// ======================================================
// STORE FLAGS
// ======================================================
GVL_CONFIG_VALIDATION.G_Config_Valid := NOT L_Config_Error;
GVL_CONFIG_VALIDATION.G_Config_Critical_Error := L_Config_Error;
GVL_CONFIG_VALIDATION.G_Config_Last_Update_MS := GVL_STATUS.G_System_Time_MS;

IF L_Config_Error THEN
    GVL_CONFIG_VALIDATION.G_Config_Last_Error_Text := 'CONFIG VALIDATION ERROR';
    GVL_STATUS.G_System_Mode_Text := 'CONFIG ERROR';
ELSE
    GVL_CONFIG_VALIDATION.G_Config_Last_Error_Text := '';
END_IF;
          
END_PROGRAM

PROGRAM PRG_Governance_Observer_Consensus_Governor
  VAR
    L_Now_MS : UDINT;
    L_Consensus_Valid : BOOL := TRUE;
    L_Error_Code : UDINT := 0;
    L_Error_Text : STRING(160) := '';
  END_VAR

            L_Now_MS := GVL_STATUS.G_System_Time_MS;
L_Consensus_Valid := TRUE;
L_Error_Code := 0;
L_Error_Text := '';

// Fail-safe defaults.
GVL_GOVERNANCE_OBSERVER_CONSENSUS_FABRIC.Governance_Observer_Consensus_Valid := FALSE;
GVL_GOVERNANCE_OBSERVER_CONSENSUS_FABRIC.Governance_Observer_Consensus_Granted := FALSE;
GVL_GOVERNANCE_OBSERVER_CONSENSUS_FABRIC.Governance_Observer_Consensus_Quarantine_Active := TRUE;

GVL_GOVERNANCE_OBSERVER_CONSENSUS_FABRIC.Distributed_Governance_Projection_Consistent := FALSE;
GVL_GOVERNANCE_OBSERVER_CONSENSUS_FABRIC.Observer_Semantic_Consensus_Valid := FALSE;
GVL_GOVERNANCE_OBSERVER_CONSENSUS_FABRIC.CrossNode_Authority_Interpretation_Aligned := FALSE;
GVL_GOVERNANCE_OBSERVER_CONSENSUS_FABRIC.Governance_Reality_Canonical := FALSE;
GVL_GOVERNANCE_OBSERVER_CONSENSUS_FABRIC.Observer_Projection_Lineage_Coherent := FALSE;

// Semantic epoch invariance required.
IF NOT GVL_SEMANTIC_EPOCH_INVARIANCE_FABRIC.Semantic_Epoch_Invariance_Granted THEN
    L_Consensus_Valid := FALSE;
    L_Error_Code := 50000;
    L_Error_Text := 'Semantic epoch invariance not granted';
END_IF;

// Governance observer split-brain detectors.
IF GVL_GOVERNANCE_OBSERVER_CONSENSUS_FABRIC.Observer_Governance_Divergence_Detected THEN
    L_Consensus_Valid := FALSE;
    L_Error_Code := 50001;
    L_Error_Text := 'Observer governance divergence detected';
END_IF;

IF GVL_GOVERNANCE_OBSERVER_CONSENSUS_FABRIC.CrossNode_Authority_Interpretation_Fork THEN
    L_Consensus_Valid := FALSE;
    L_Error_Code := 50002;
    L_Error_Text := 'Cross-node authority interpretation fork detected';
END_IF;

IF GVL_GOVERNANCE_OBSERVER_CONSENSUS_FABRIC.Semantic_Projection_Mismatch_Detected THEN
    L_Consensus_Valid := FALSE;
    L_Error_Code := 50003;
    L_Error_Text := 'Semantic projection mismatch detected';
END_IF;

IF GVL_GOVERNANCE_OBSERVER_CONSENSUS_FABRIC.Canonical_Governance_Reality_Lost THEN
    L_Consensus_Valid := FALSE;
    L_Error_Code := 50004;
    L_Error_Text := 'Canonical governance reality lost';
END_IF;

IF GVL_GOVERNANCE_OBSERVER_CONSENSUS_FABRIC.Observer_Projection_Lineage_Drift_Detected THEN
    L_Consensus_Valid := FALSE;
    L_Error_Code := 50005;
    L_Error_Text := 'Observer projection lineage drift detected';
END_IF;

IF GVL_GOVERNANCE_OBSERVER_CONSENSUS_FABRIC.Distributed_Governance_Reality_Fork_Detected THEN
    L_Consensus_Valid := FALSE;
    L_Error_Code := 50006;
    L_Error_Text := 'Distributed governance reality fork detected';
END_IF;

// Observer consensus validation.
IF L_Consensus_Valid
AND NOT GVL_GOVERNANCE_OBSERVER_CONSENSUS_FABRIC.Canonical_Projection_Vector_Stable THEN
    L_Consensus_Valid := FALSE;
    L_Error_Code := 50010;
    L_Error_Text := 'Canonical projection vector invalid';
END_IF;

IF L_Consensus_Valid
AND NOT GVL_GOVERNANCE_OBSERVER_CONSENSUS_FABRIC.Distributed_Interpretation_Equivalence_Valid THEN
    L_Consensus_Valid := FALSE;
    L_Error_Code := 50011;
    L_Error_Text := 'Distributed interpretation equivalence invalid';
END_IF;

IF L_Consensus_Valid
AND NOT GVL_GOVERNANCE_OBSERVER_CONSENSUS_FABRIC.Governance_Projection_Causality_Grounded THEN
    L_Consensus_Valid := FALSE;
    L_Error_Code := 50012;
    L_Error_Text := 'Governance projection causality invalid';
END_IF;

IF L_Consensus_Valid
AND NOT GVL_GOVERNANCE_OBSERVER_CONSENSUS_FABRIC.Observer_Timeline_Consensus_Monotonic THEN
    L_Consensus_Valid := FALSE;
    L_Error_Code := 50013;
    L_Error_Text := 'Observer timeline consensus monotonicity invalid';
END_IF;

IF L_Consensus_Valid THEN
    GVL_GOVERNANCE_OBSERVER_CONSENSUS_FABRIC.Governance_Observer_Consensus_Valid := TRUE;
    GVL_GOVERNANCE_OBSERVER_CONSENSUS_FABRIC.Governance_Observer_Consensus_Granted := TRUE;
    GVL_GOVERNANCE_OBSERVER_CONSENSUS_FABRIC.Governance_Observer_Consensus_Quarantine_Active := FALSE;

    GVL_GOVERNANCE_OBSERVER_CONSENSUS_FABRIC.Distributed_Governance_Projection_Consistent := TRUE;
    GVL_GOVERNANCE_OBSERVER_CONSENSUS_FABRIC.Observer_Semantic_Consensus_Valid := TRUE;
    GVL_GOVERNANCE_OBSERVER_CONSENSUS_FABRIC.CrossNode_Authority_Interpretation_Aligned := TRUE;
    GVL_GOVERNANCE_OBSERVER_CONSENSUS_FABRIC.Governance_Reality_Canonical := TRUE;
    GVL_GOVERNANCE_OBSERVER_CONSENSUS_FABRIC.Observer_Projection_Lineage_Coherent := TRUE;

    GVL_GOVERNANCE_OBSERVER_CONSENSUS_FABRIC.Governance_Observer_Consensus_Epoch :=
        GVL_SEMANTIC_EPOCH_INVARIANCE_FABRIC.Semantic_Epoch_Invariance_Epoch;

    GVL_GOVERNANCE_OBSERVER_CONSENSUS_FABRIC.Governance_Observer_Consensus_Epoch_Coherent := TRUE;

    GVL_GOVERNANCE_OBSERVER_CONSENSUS_FABRIC.Governance_Observer_Consensus_Last_Update_MS :=
        L_Now_MS;

    GVL_GOVERNANCE_OBSERVER_CONSENSUS_FABRIC.Governance_Observer_Consensus_Lease_Expired := FALSE;

    GVL_GOVERNANCE_OBSERVER_CONSENSUS_FABRIC.Governance_Observer_Consensus_Last_Error_Code := 0;
    GVL_GOVERNANCE_OBSERVER_CONSENSUS_FABRIC.Governance_Observer_Consensus_Last_Error_Text := '';
ELSE
    GVL_GOVERNANCE_OBSERVER_CONSENSUS_FABRIC.Governance_Observer_Consensus_Valid := FALSE;
    GVL_GOVERNANCE_OBSERVER_CONSENSUS_FABRIC.Governance_Observer_Consensus_Granted := FALSE;
    GVL_GOVERNANCE_OBSERVER_CONSENSUS_FABRIC.Governance_Observer_Consensus_Quarantine_Active := TRUE;

    GVL_GOVERNANCE_OBSERVER_CONSENSUS_FABRIC.Governance_Observer_Consensus_Lease_Expired := TRUE;

    GVL_GOVERNANCE_OBSERVER_CONSENSUS_FABRIC.Governance_Observer_Consensus_Last_Error_Code :=
        L_Error_Code;

    GVL_GOVERNANCE_OBSERVER_CONSENSUS_FABRIC.Governance_Observer_Consensus_Last_Error_Text :=
        L_Error_Text;

    GVL_GOVERNANCE_OBSERVER_CONSENSUS_FABRIC.Governance_Observer_Consensus_Invalidation_Count :=
        GVL_GOVERNANCE_OBSERVER_CONSENSUS_FABRIC.Governance_Observer_Consensus_Invalidation_Count + 1;
END_IF;
          
END_PROGRAM

PROGRAM PRG_Transport_Freshness_Governor
  VAR
    L_Now_MS : UDINT;
    L_Delta_MS : UDINT;
    L_Transport_Valid : BOOL := TRUE;
    L_Error_Code : UDINT := 0;
    L_Error_Text : STRING(160) := '';
  END_VAR

            L_Now_MS := GVL_STATUS.G_System_Time_MS;
L_Transport_Valid := TRUE;
L_Error_Code := 0;
L_Error_Text := '';

// ======================================================
// TRANSPORT FRESHNESS GOVERNOR
// ======================================================
// Governs transport freshness semantics.
// Prevents stale transport semantic publication.
//
// Transport freshness is upstream of runtime barrier in MAIN.
// It must not consume runtime barrier or downstream recovery
// governance state, because runtime barrier consumes transport
// freshness state later in the same scan-cycle.
// ======================================================

GVL_TRANSPORT_FRESHNESS.Transport_Stale_Frame_Detected := FALSE;
GVL_TRANSPORT_FRESHNESS.Transport_Transaction_Mismatch := FALSE;
GVL_TRANSPORT_FRESHNESS.Transport_Snapshot_Invalid := FALSE;

// Monotonic authority linkage.
IF L_Transport_Valid AND (NOT GVL_TIME_MONOTONIC.Monotonic_Time_Valid) THEN
    L_Transport_Valid := FALSE;
    L_Error_Code := 10001;
    L_Error_Text := 'Transport monotonic authority invalid';
END_IF;

// Transport reconnect quarantine.
IF GVL_TRANSPORT_FRESHNESS.Transport_Reconnect_Stabilizing THEN
    GVL_TRANSPORT_FRESHNESS.Transport_Quarantine_Active := TRUE;

    L_Transport_Valid := FALSE;

    IF L_Error_Code = 0 THEN
        L_Error_Code := 10003;
        L_Error_Text := 'Transport reconnect stabilization active';
    END_IF;
END_IF;

// Lease freshness validation.
L_Delta_MS := L_Now_MS - GVL_TRANSPORT_FRESHNESS.Transport_Last_Refresh_MS;

IF L_Transport_Valid AND GVL_TRANSPORT_FRESHNESS.Transport_Lease_Valid THEN
    IF L_Delta_MS > GVL_TRANSPORT_FRESHNESS.Transport_Lease_Timeout_MS THEN
        L_Transport_Valid := FALSE;
        L_Error_Code := 10004;
        L_Error_Text := 'Transport lease expired';

        GVL_TRANSPORT_FRESHNESS.Transport_Lease_Expired := TRUE;
    END_IF;
END_IF;

// Publish authoritative transport freshness state.
IF L_Transport_Valid THEN
    GVL_TRANSPORT_FRESHNESS.Transport_Epoch := GVL_TRANSPORT_FRESHNESS.Transport_Epoch + 1;
    GVL_TRANSPORT_FRESHNESS.Transport_Publication_Epoch := GVL_TRANSPORT_FRESHNESS.Transport_Publication_Epoch + 1;

    GVL_TRANSPORT_FRESHNESS.Transport_Freshness_Valid := TRUE;
    GVL_TRANSPORT_FRESHNESS.Transport_Publication_Allowed := TRUE;

    GVL_TRANSPORT_FRESHNESS.Transport_Lease_Valid := TRUE;
    GVL_TRANSPORT_FRESHNESS.Transport_Lease_Expired := FALSE;

    GVL_TRANSPORT_FRESHNESS.Transport_Quarantine_Active := FALSE;

    GVL_TRANSPORT_FRESHNESS.Transport_Last_Refresh_MS := L_Now_MS;
    GVL_TRANSPORT_FRESHNESS.Transport_Last_Publication_MS := L_Now_MS;

    GVL_TRANSPORT_FRESHNESS.Transport_Last_Error_Code := 0;
    GVL_TRANSPORT_FRESHNESS.Transport_Last_Error_Text := '';
ELSE
    GVL_TRANSPORT_FRESHNESS.Transport_Freshness_Valid := FALSE;
    GVL_TRANSPORT_FRESHNESS.Transport_Publication_Allowed := FALSE;

    GVL_TRANSPORT_FRESHNESS.Transport_Snapshot_Invalid := TRUE;

    GVL_TRANSPORT_FRESHNESS.Transport_Last_Error_Code := L_Error_Code;
    GVL_TRANSPORT_FRESHNESS.Transport_Last_Error_Text := L_Error_Text;

    GVL_TRANSPORT_FRESHNESS.Transport_Invalidation_Count := GVL_TRANSPORT_FRESHNESS.Transport_Invalidation_Count + 1;
END_IF;
          
END_PROGRAM

PROGRAM PRG_Semantic_Epoch_Invariance_Governor
  VAR
    L_Now_MS : UDINT;
    L_Invariance_Valid : BOOL := TRUE;
    L_Error_Code : UDINT := 0;
    L_Error_Text : STRING(160) := '';
  END_VAR

            L_Now_MS := GVL_STATUS.G_System_Time_MS;
L_Invariance_Valid := TRUE;
L_Error_Code := 0;
L_Error_Text := '';

// Fail-safe defaults.
GVL_SEMANTIC_EPOCH_INVARIANCE_FABRIC.Semantic_Epoch_Invariance_Valid := FALSE;
GVL_SEMANTIC_EPOCH_INVARIANCE_FABRIC.Semantic_Epoch_Invariance_Granted := FALSE;
GVL_SEMANTIC_EPOCH_INVARIANCE_FABRIC.Semantic_Epoch_Invariance_Quarantine_Active := TRUE;

GVL_SEMANTIC_EPOCH_INVARIANCE_FABRIC.Authority_Semantics_Invariant := FALSE;
GVL_SEMANTIC_EPOCH_INVARIANCE_FABRIC.CrossEpoch_Permission_Mapping_Stable := FALSE;
GVL_SEMANTIC_EPOCH_INVARIANCE_FABRIC.Semantic_Intent_Continuity_Valid := FALSE;
GVL_SEMANTIC_EPOCH_INVARIANCE_FABRIC.Governance_Meaning_Preservation_Coherent := FALSE;
GVL_SEMANTIC_EPOCH_INVARIANCE_FABRIC.Semantic_Evolution_Lineage_Traceable := FALSE;

// Trust epoch monotonicity required.
IF NOT GVL_TRUST_EPOCH_MONOTONICITY_FABRIC.Trust_Epoch_Monotonicity_Granted THEN
    L_Invariance_Valid := FALSE;
    L_Error_Code := 49000;
    L_Error_Text := 'Trust epoch monotonicity not granted';
END_IF;

// Semantic epoch drift detectors.
IF GVL_SEMANTIC_EPOCH_INVARIANCE_FABRIC.Semantic_Authority_Drift_Detected THEN
    L_Invariance_Valid := FALSE;
    L_Error_Code := 49001;
    L_Error_Text := 'Semantic authority drift detected';
END_IF;

IF GVL_SEMANTIC_EPOCH_INVARIANCE_FABRIC.CrossEpoch_Permission_Reinterpretation THEN
    L_Invariance_Valid := FALSE;
    L_Error_Code := 49002;
    L_Error_Text := 'Cross-epoch permission reinterpretation detected';
END_IF;

IF GVL_SEMANTIC_EPOCH_INVARIANCE_FABRIC.Intent_To_Authority_Mismatch_Detected THEN
    L_Invariance_Valid := FALSE;
    L_Error_Code := 49003;
    L_Error_Text := 'Intent-to-authority mismatch detected';
END_IF;

IF GVL_SEMANTIC_EPOCH_INVARIANCE_FABRIC.Governance_Semantic_Fork_Detected THEN
    L_Invariance_Valid := FALSE;
    L_Error_Code := 49004;
    L_Error_Text := 'Governance semantic fork detected';
END_IF;

IF GVL_SEMANTIC_EPOCH_INVARIANCE_FABRIC.Semantic_Migration_Lineage_Gap_Detected THEN
    L_Invariance_Valid := FALSE;
    L_Error_Code := 49005;
    L_Error_Text := 'Semantic migration lineage gap detected';
END_IF;

IF GVL_SEMANTIC_EPOCH_INVARIANCE_FABRIC.Distributed_Semantic_Divergence_Detected THEN
    L_Invariance_Valid := FALSE;
    L_Error_Code := 49006;
    L_Error_Text := 'Distributed semantic divergence detected';
END_IF;

// Semantic invariance validation.
IF L_Invariance_Valid
AND NOT GVL_SEMANTIC_EPOCH_INVARIANCE_FABRIC.Explicit_Semantic_Migration_Governed THEN
    L_Invariance_Valid := FALSE;
    L_Error_Code := 49010;
    L_Error_Text := 'Explicit semantic migration governance invalid';
END_IF;

IF L_Invariance_Valid
AND NOT GVL_SEMANTIC_EPOCH_INVARIANCE_FABRIC.CrossEpoch_Semantic_Equivalence_Valid THEN
    L_Invariance_Valid := FALSE;
    L_Error_Code := 49011;
    L_Error_Text := 'Cross-epoch semantic equivalence invalid';
END_IF;

IF L_Invariance_Valid
AND NOT GVL_SEMANTIC_EPOCH_INVARIANCE_FABRIC.Distributed_Semantic_Consensus_Stable THEN
    L_Invariance_Valid := FALSE;
    L_Error_Code := 49012;
    L_Error_Text := 'Distributed semantic consensus invalid';
END_IF;

IF L_Invariance_Valid
AND NOT GVL_SEMANTIC_EPOCH_INVARIANCE_FABRIC.Semantic_Interpretation_Integrity_Valid THEN
    L_Invariance_Valid := FALSE;
    L_Error_Code := 49013;
    L_Error_Text := 'Semantic interpretation integrity invalid';
END_IF;

IF L_Invariance_Valid THEN
    GVL_SEMANTIC_EPOCH_INVARIANCE_FABRIC.Semantic_Epoch_Invariance_Valid := TRUE;
    GVL_SEMANTIC_EPOCH_INVARIANCE_FABRIC.Semantic_Epoch_Invariance_Granted := TRUE;
    GVL_SEMANTIC_EPOCH_INVARIANCE_FABRIC.Semantic_Epoch_Invariance_Quarantine_Active := FALSE;

    GVL_SEMANTIC_EPOCH_INVARIANCE_FABRIC.Authority_Semantics_Invariant := TRUE;
    GVL_SEMANTIC_EPOCH_INVARIANCE_FABRIC.CrossEpoch_Permission_Mapping_Stable := TRUE;
    GVL_SEMANTIC_EPOCH_INVARIANCE_FABRIC.Semantic_Intent_Continuity_Valid := TRUE;
    GVL_SEMANTIC_EPOCH_INVARIANCE_FABRIC.Governance_Meaning_Preservation_Coherent := TRUE;
    GVL_SEMANTIC_EPOCH_INVARIANCE_FABRIC.Semantic_Evolution_Lineage_Traceable := TRUE;

    GVL_SEMANTIC_EPOCH_INVARIANCE_FABRIC.Semantic_Epoch_Invariance_Epoch :=
        GVL_TRUST_EPOCH_MONOTONICITY_FABRIC.Trust_Epoch_Monotonicity_Epoch;

    GVL_SEMANTIC_EPOCH_INVARIANCE_FABRIC.Semantic_Epoch_Invariance_Epoch_Coherent := TRUE;

    GVL_SEMANTIC_EPOCH_INVARIANCE_FABRIC.Semantic_Epoch_Invariance_Last_Update_MS :=
        L_Now_MS;

    GVL_SEMANTIC_EPOCH_INVARIANCE_FABRIC.Semantic_Epoch_Invariance_Lease_Expired := FALSE;

    GVL_SEMANTIC_EPOCH_INVARIANCE_FABRIC.Semantic_Epoch_Invariance_Last_Error_Code := 0;
    GVL_SEMANTIC_EPOCH_INVARIANCE_FABRIC.Semantic_Epoch_Invariance_Last_Error_Text := '';
ELSE
    GVL_SEMANTIC_EPOCH_INVARIANCE_FABRIC.Semantic_Epoch_Invariance_Valid := FALSE;
    GVL_SEMANTIC_EPOCH_INVARIANCE_FABRIC.Semantic_Epoch_Invariance_Granted := FALSE;
    GVL_SEMANTIC_EPOCH_INVARIANCE_FABRIC.Semantic_Epoch_Invariance_Quarantine_Active := TRUE;

    GVL_SEMANTIC_EPOCH_INVARIANCE_FABRIC.Semantic_Epoch_Invariance_Lease_Expired := TRUE;

    GVL_SEMANTIC_EPOCH_INVARIANCE_FABRIC.Semantic_Epoch_Invariance_Last_Error_Code :=
        L_Error_Code;

    GVL_SEMANTIC_EPOCH_INVARIANCE_FABRIC.Semantic_Epoch_Invariance_Last_Error_Text :=
        L_Error_Text;

    GVL_SEMANTIC_EPOCH_INVARIANCE_FABRIC.Semantic_Epoch_Invariance_Invalidation_Count :=
        GVL_SEMANTIC_EPOCH_INVARIANCE_FABRIC.Semantic_Epoch_Invariance_Invalidation_Count + 1;
END_IF;
          
END_PROGRAM

PROGRAM PRG_Scenario_Engine
  VAR
    L_Hour : INT;
    L_Hum : REAL;
    L_ZoneWeight : REAL;
    L_AdaptConfidence : REAL;
    L_InputConfidence : REAL;
    L_ZoneConfidence : REAL;
    L_ZoneScore : REAL;
    L_BestVentScore : REAL;
    L_BestVentZone : INT;
    L_i : INT;
    fbTrace : FB_Trace_Write;
    L_Weights : ST_Behavior_Weights;
  END_VAR

            // Build weights from compile-safe scalar GVL fields
L_Weights.W_Comfort := GVL_BEHAVIOR_ADAPT.G_Behavior_Weight_Comfort;
L_Weights.W_Night := GVL_BEHAVIOR_ADAPT.G_Behavior_Weight_Night;
L_Weights.W_Preheat := GVL_BEHAVIOR_ADAPT.G_Behavior_Weight_Preheat;
L_Weights.W_VentBoost := GVL_BEHAVIOR_ADAPT.G_Behavior_Weight_VentBoost;
L_Weights.W_AccessSecure := GVL_BEHAVIOR_ADAPT.G_Behavior_Weight_AccessSecure;

L_Hour := TO_INT(GVL_TIME_SERVICE.G_Time_Of_Day_MS / 3600000);

// Reset
GVL_INTENT_BEHAVIOR.I_Request_Night_Mode := FALSE;
GVL_INTENT_BEHAVIOR.I_Request_Comfort_Mode := FALSE;
GVL_INTENT_BEHAVIOR.I_Request_Ventilation_Boost := FALSE;
GVL_INTENT_BEHAVIOR.I_Request_Access_Secure_Mode := FALSE;

GVL_INTENT_BEHAVIOR.I_Score_Comfort := REAL_TO_INT(GVL_SCENARIO_CONFIG.G_Comfort_Base_Score * L_Weights.W_Comfort);
GVL_INTENT_BEHAVIOR.I_Score_Night := 0;
GVL_INTENT_BEHAVIOR.I_Score_Preheat := 0;
GVL_INTENT_BEHAVIOR.I_Score_Vent_Boost := 0;
GVL_INTENT_BEHAVIOR.I_Score_Access_Secure := 0;

// Night
IF (L_Hour >= GVL_SCENARIO_CONFIG.G_Night_Start_Hour) OR (L_Hour < GVL_SCENARIO_CONFIG.G_Night_End_Hour) THEN
    GVL_INTENT_BEHAVIOR.I_Score_Night := REAL_TO_INT(GVL_SCENARIO_CONFIG.G_Night_Base_Score * L_Weights.W_Night);
END_IF;

// Preheat
IF GVL_INPUT.IN_Preheat_Request THEN
    GVL_INTENT_BEHAVIOR.I_Score_Preheat := REAL_TO_INT(GVL_SCENARIO_CONFIG.G_Preheat_Base_Score * L_Weights.W_Preheat);
END_IF;

// Vent boost
L_BestVentScore := 0.0;
L_BestVentZone := 0;

FOR L_i := 1 TO GVL_CONSTANTS.C_MAX_ZONES DO
    L_Hum := GVL_INPUT.IN_Room_Hum[L_i];

    IF GVL_BEHAVIOR_ADAPT.G_VentBoost_Zone_Adapt[L_i].Zone_Weight = 0.0 THEN
        L_ZoneWeight := GVL_BEHAVIOR_ADAPT.G_Adapt_Default_Zone_Weight;
    ELSE
        L_ZoneWeight := GVL_BEHAVIOR_ADAPT.G_VentBoost_Zone_Adapt[L_i].Zone_Weight;
    END_IF;

    L_AdaptConfidence := GVL_BEHAVIOR_ADAPT.G_VentBoost_Zone_Adapt[L_i].Confidence;
    IF L_AdaptConfidence <= 0.0 THEN
        L_AdaptConfidence := GVL_SCENARIO_CONFIG.G_Fallback_Adapt_Confidence;
    END_IF;

    L_InputConfidence := GVL_INPUT.IN_Zone_Confidence[L_i];
    IF L_InputConfidence <= 0.0 THEN
        L_InputConfidence := GVL_SCENARIO_CONFIG.G_Fallback_Input_Confidence;
    END_IF;

    L_ZoneConfidence := L_AdaptConfidence * L_InputConfidence;

    IF L_Hum > GVL_SCENARIO_CONFIG.G_VentBoost_Humidity_Threshold THEN
        L_ZoneScore := GVL_SCENARIO_CONFIG.G_VentBoost_Base_Score * L_Weights.W_VentBoost * L_ZoneWeight * L_ZoneConfidence;

        IF L_ZoneScore > L_BestVentScore THEN
            L_BestVentScore := L_ZoneScore;
            L_BestVentZone := L_i;
        END_IF;
    END_IF;
END_FOR;

GVL_INTENT_BEHAVIOR.I_Score_Vent_Boost := REAL_TO_INT(L_BestVentScore);
GVL_INTENT_BEHAVIOR.I_Best_VentBoost_Zone := L_BestVentZone;

// Access secure
IF (L_Hour >= GVL_SCENARIO_CONFIG.G_Access_Secure_Start_Hour) OR (L_Hour < GVL_SCENARIO_CONFIG.G_Access_Secure_End_Hour) THEN
    GVL_INTENT_BEHAVIOR.I_Score_Access_Secure := REAL_TO_INT(GVL_SCENARIO_CONFIG.G_AccessSecure_Base_Score * L_Weights.W_AccessSecure);
END_IF;

// Activate flags
IF GVL_INTENT_BEHAVIOR.I_Score_Night >= GVL_SCENARIO_CONFIG.G_Night_Activation_Threshold THEN
    GVL_INTENT_BEHAVIOR.I_Request_Night_Mode := TRUE;
END_IF;

IF GVL_INTENT_BEHAVIOR.I_Score_Preheat >= GVL_SCENARIO_CONFIG.G_Comfort_Activation_Threshold THEN
    GVL_INTENT_BEHAVIOR.I_Request_Comfort_Mode := TRUE;
END_IF;

IF GVL_INTENT_BEHAVIOR.I_Score_Vent_Boost >= GVL_SCENARIO_CONFIG.G_VentBoost_Activation_Threshold THEN
    GVL_INTENT_BEHAVIOR.I_Request_Ventilation_Boost := TRUE;
END_IF;

IF GVL_INTENT_BEHAVIOR.I_Score_Access_Secure >= GVL_SCENARIO_CONFIG.G_AccessSecure_Activation_Threshold THEN
    GVL_INTENT_BEHAVIOR.I_Request_Access_Secure_Mode := TRUE;
END_IF;

// Multi-objective weights
GVL_INTENT_BEHAVIOR.I_Weight_Night := TO_REAL(GVL_INTENT_BEHAVIOR.I_Score_Night) / 100.0;
GVL_INTENT_BEHAVIOR.I_Weight_Comfort := TO_REAL(GVL_INTENT_BEHAVIOR.I_Score_Comfort) / 100.0;
GVL_INTENT_BEHAVIOR.I_Weight_Vent_Boost := TO_REAL(GVL_INTENT_BEHAVIOR.I_Score_Vent_Boost) / 100.0;
GVL_INTENT_BEHAVIOR.I_Weight_Access_Secure := TO_REAL(GVL_INTENT_BEHAVIOR.I_Score_Access_Secure) / 100.0;

// Scenario text
IF GVL_INTENT_BEHAVIOR.I_Request_Night_Mode THEN
    GVL_INTENT_BEHAVIOR.I_Selected_Scenario_Text := 'Night mode';
ELSIF GVL_INTENT_BEHAVIOR.I_Request_Ventilation_Boost THEN
    GVL_INTENT_BEHAVIOR.I_Selected_Scenario_Text := 'Vent Boost';
ELSIF GVL_INTENT_BEHAVIOR.I_Request_Comfort_Mode THEN
    GVL_INTENT_BEHAVIOR.I_Selected_Scenario_Text := 'Comfort';
ELSIF GVL_INTENT_BEHAVIOR.I_Request_Access_Secure_Mode THEN
    GVL_INTENT_BEHAVIOR.I_Selected_Scenario_Text := 'Access Secure';
ELSE
    GVL_INTENT_BEHAVIOR.I_Selected_Scenario_Text := 'Idle';
END_IF;

GVL_INTENT_BEHAVIOR.I_Reason_Text := GVL_INTENT_BEHAVIOR.I_Selected_Scenario_Text;
GVL_INTENT_BEHAVIOR.I_Last_Update_MS := GVL_TIME_SERVICE.G_Now_MS;

fbTrace(iLayer:=TRACE_SCENARIO,iSource:=SRC_SCENARIO,iReason:=REASON_SCENARIO_VENT_BOOST,iValueBool:=GVL_INTENT_BEHAVIOR.I_Request_Ventilation_Boost,iValueReal:=TO_REAL(GVL_INTENT_BEHAVIOR.I_Score_Vent_Boost),iText:=GVL_INTENT_BEHAVIOR.I_Selected_Scenario_Text);
          
END_PROGRAM

PROGRAM PRG_Distributed_Peer_Ingestion
  VAR
    L_Now_MS : UDINT;
  END_VAR

            // ======================================================
// DISTRIBUTED PEER INGESTION
// ======================================================
// Bounded peer-session ingestion layer.
//
// Purpose:
// normalize replicated HA session state into distributed
// peer-input fields consumed by distributed governors.
//
// This layer does NOT:
// - perform reconciliation/quarantine decisions
// - perform split-brain detection
// - validate peer publication correctness
// - mutate local runtime authority
// ======================================================

L_Now_MS := GVL_STATUS.G_System_Time_MS;

// ------------------------------------------------------
// Peer session freshness projection.
// ------------------------------------------------------

GVL_DISTRIBUTED_EPOCH.Peer_Last_Refresh_MS :=
    GVL_HA_SESSION_REPLICATION.HA_Remote_Last_Refresh_MS;

GVL_DISTRIBUTED_EPOCH.Peer_Lease_Active :=
    GVL_HA_SESSION_REPLICATION.HA_Remote_Session_Valid;

// ------------------------------------------------------
// Replicated remote session ingestion.
// ------------------------------------------------------

IF GVL_HA_SESSION_REPLICATION.HA_Remote_Session_Valid THEN
    GVL_DISTRIBUTED_EPOCH.Peer_Runtime_Epoch :=
        GVL_HA_SESSION_REPLICATION.HA_Remote_Runtime_Epoch;

    GVL_DISTRIBUTED_EPOCH.Peer_Snapshot_Epoch :=
        GVL_HA_SESSION_REPLICATION.HA_Remote_Snapshot_Epoch;

    GVL_DISTRIBUTED_EPOCH.Peer_Boot_Generation :=
        GVL_HA_SESSION_REPLICATION.HA_Remote_Boot_Generation;

    GVL_DISTRIBUTED_EPOCH.Peer_Fencing_Token :=
        GVL_HA_SESSION_REPLICATION.HA_Remote_Fencing_Token;
ELSE
    GVL_DISTRIBUTED_EPOCH.Peer_Lease_Active := FALSE;
    GVL_DISTRIBUTED_EPOCH.Peer_Runtime_Epoch := 0;
    GVL_DISTRIBUTED_EPOCH.Peer_Snapshot_Epoch := 0;
    GVL_DISTRIBUTED_EPOCH.Peer_Boot_Generation := 0;
    GVL_DISTRIBUTED_EPOCH.Peer_Fencing_Token := 0;
    GVL_DISTRIBUTED_EPOCH.Peer_Last_Refresh_MS := 0;
END_IF;

// >>> BULK_SYNC_ANCHOR: PRG_Distributed_Peer_Ingestion <<<
          
END_PROGRAM

PROGRAM PRG_Industrial_Maintainability_Governor

            // Passive maintainability governance placeholder.
// Runtime maintainability state is currently represented by fabric GVLs only.
// This program is intentionally side-effect free until ownership is formalized.
          
END_PROGRAM

PROGRAM PRG_Sensor_Consensus_Governor
  VAR
    L_Now_MS : UDINT;
    L_Consensus_Valid : BOOL := TRUE;
    L_Error_Code : UDINT := 0;
    L_Error_Text : STRING(160) := '';
    L_Consensus_Age_MS : UDINT;
  END_VAR

            L_Now_MS := GVL_STATUS.G_System_Time_MS;
L_Consensus_Valid := TRUE;
L_Error_Code := 0;
L_Error_Text := '';

// Fail-safe defaults.
GVL_SENSOR_CONSENSUS.Sensor_Consensus_Valid := FALSE;
GVL_SENSOR_CONSENSUS.Sensor_Consensus_Quarantine_Active := TRUE;
GVL_SENSOR_CONSENSUS.Sensor_Consensus_Lease_Expired := TRUE;
GVL_SENSOR_CONSENSUS.Sensor_Consensus_Freshness_Valid := FALSE;

GVL_SENSOR_CONSENSUS.Physics_Invariants_Satisfied := FALSE;
GVL_SENSOR_CONSENSUS.Cross_Sensor_Correlation_Valid := FALSE;
GVL_SENSOR_CONSENSUS.Telemetry_Plausibility_Valid := FALSE;

IF GVL_SENSOR_CONSENSUS.Sensor_Replay_Suspected THEN
    L_Consensus_Valid := FALSE;
    L_Error_Code := 22000;
    L_Error_Text := 'Sensor replay suspected';
END_IF;

IF L_Consensus_Valid
AND GVL_SENSOR_CONSENSUS.Sensor_Partition_Detected THEN
    L_Consensus_Valid := FALSE;
    L_Error_Code := 22001;
    L_Error_Text := 'Sensor partition detected';
END_IF;

IF L_Consensus_Valid
AND GVL_SENSOR_CONSENSUS.Sensor_Hallucination_Suspected THEN
    L_Consensus_Valid := FALSE;
    L_Error_Code := 22002;
    L_Error_Text := 'Sensor hallucination suspected';
END_IF;

IF L_Consensus_Valid
AND GVL_SENSOR_CONSENSUS.Cross_Sensor_Divergence_Detected THEN
    L_Consensus_Valid := FALSE;
    L_Error_Code := 22003;
    L_Error_Text := 'Cross sensor divergence detected';
END_IF;

IF L_Consensus_Valid
AND GVL_SENSOR_CONSENSUS.Sensor_Drift_Detected THEN
    L_Consensus_Valid := FALSE;
    L_Error_Code := 22004;
    L_Error_Text := 'Sensor drift detected';
END_IF;

IF L_Consensus_Valid
AND GVL_SENSOR_CONSENSUS.Sensor_Oscillation_Detected THEN
    L_Consensus_Valid := FALSE;
    L_Error_Code := 22005;
    L_Error_Text := 'Sensor oscillation detected';
END_IF;

IF L_Consensus_Valid
AND GVL_SENSOR_CONSENSUS.Sensor_Stuck_State_Detected THEN
    L_Consensus_Valid := FALSE;
    L_Error_Code := 22006;
    L_Error_Text := 'Sensor stuck state detected';
END_IF;

// Physics invariants.
IF L_Consensus_Valid
AND NOT GVL_SENSOR_CONSENSUS.Flow_Response_Valid THEN
    L_Consensus_Valid := FALSE;
    L_Error_Code := 22010;
    L_Error_Text := 'Flow response invalid';
END_IF;

IF L_Consensus_Valid
AND NOT GVL_SENSOR_CONSENSUS.Pressure_Response_Valid THEN
    L_Consensus_Valid := FALSE;
    L_Error_Code := 22011;
    L_Error_Text := 'Pressure response invalid';
END_IF;

IF L_Consensus_Valid
AND NOT GVL_SENSOR_CONSENSUS.Airflow_Response_Valid THEN
    L_Consensus_Valid := FALSE;
    L_Error_Code := 22012;
    L_Error_Text := 'Airflow response invalid';
END_IF;

IF L_Consensus_Valid
AND NOT GVL_SENSOR_CONSENSUS.Current_Signature_Valid THEN
    L_Consensus_Valid := FALSE;
    L_Error_Code := 22013;
    L_Error_Text := 'Current signature invalid';
END_IF;

// Consensus freshness.
L_Consensus_Age_MS :=
    L_Now_MS - GVL_SENSOR_CONSENSUS.Last_Consensus_Update_MS;

IF L_Consensus_Valid
AND (L_Consensus_Age_MS > 5000) THEN
    L_Consensus_Valid := FALSE;
    L_Error_Code := 22020;
    L_Error_Text := 'Sensor consensus stale';
END_IF;

IF L_Consensus_Valid THEN
    GVL_SENSOR_CONSENSUS.Sensor_Consensus_Valid := TRUE;
    GVL_SENSOR_CONSENSUS.Sensor_Consensus_Quarantine_Active := FALSE;
    GVL_SENSOR_CONSENSUS.Sensor_Consensus_Lease_Expired := FALSE;
    GVL_SENSOR_CONSENSUS.Sensor_Consensus_Freshness_Valid := TRUE;

    GVL_SENSOR_CONSENSUS.Physics_Invariants_Satisfied := TRUE;
    GVL_SENSOR_CONSENSUS.Cross_Sensor_Correlation_Valid := TRUE;
    GVL_SENSOR_CONSENSUS.Telemetry_Plausibility_Valid := TRUE;

    GVL_SENSOR_CONSENSUS.Sensor_Consensus_Epoch :=
        GVL_SENSOR_CONSENSUS.Sensor_Consensus_Epoch + 1;

    GVL_SENSOR_CONSENSUS.Last_Consensus_Update_MS := L_Now_MS;

    GVL_SENSOR_CONSENSUS.Sensor_Consensus_Last_Error_Code := 0;
    GVL_SENSOR_CONSENSUS.Sensor_Consensus_Last_Error_Text := '';
ELSE
    GVL_SENSOR_CONSENSUS.Sensor_Consensus_Valid := FALSE;
    GVL_SENSOR_CONSENSUS.Sensor_Consensus_Quarantine_Active := TRUE;
    GVL_SENSOR_CONSENSUS.Sensor_Consensus_Lease_Expired := TRUE;
    GVL_SENSOR_CONSENSUS.Sensor_Consensus_Freshness_Valid := FALSE;

    GVL_SENSOR_CONSENSUS.Sensor_Consensus_Last_Error_Code := L_Error_Code;
    GVL_SENSOR_CONSENSUS.Sensor_Consensus_Last_Error_Text := L_Error_Text;

    GVL_SENSOR_CONSENSUS.Sensor_Consensus_Invalidation_Count :=
        GVL_SENSOR_CONSENSUS.Sensor_Consensus_Invalidation_Count + 1;
END_IF;
          
END_PROGRAM

PROGRAM PRG_Governance_Feedback_Integrity_Governor
  VAR
    L_Now_MS : UDINT;
    L_Integrity_Valid : BOOL := TRUE;
    L_Error_Code : UDINT := 0;
    L_Error_Text : STRING(160) := '';
  END_VAR

            L_Now_MS := GVL_STATUS.G_System_Time_MS;
L_Integrity_Valid := TRUE;
L_Error_Code := 0;
L_Error_Text := '';

// Fail-safe defaults.
GVL_GOVERNANCE_FEEDBACK_INTEGRITY_FABRIC.Governance_Feedback_Integrity_Valid := FALSE;
GVL_GOVERNANCE_FEEDBACK_INTEGRITY_FABRIC.Governance_Feedback_Integrity_Granted := FALSE;
GVL_GOVERNANCE_FEEDBACK_INTEGRITY_FABRIC.Governance_Feedback_Integrity_Quarantine_Active := TRUE;

GVL_GOVERNANCE_FEEDBACK_INTEGRITY_FABRIC.Execution_Feedback_Causality_Isolated := FALSE;
GVL_GOVERNANCE_FEEDBACK_INTEGRITY_FABRIC.Governance_Derivation_Inputs_Canonical := FALSE;
GVL_GOVERNANCE_FEEDBACK_INTEGRITY_FABRIC.Telemetry_To_Authority_Lineage_Valid := FALSE;
GVL_GOVERNANCE_FEEDBACK_INTEGRITY_FABRIC.Feedback_Epoch_Integrity_Stable := FALSE;
GVL_GOVERNANCE_FEEDBACK_INTEGRITY_FABRIC.Governance_Feedback_Lineage_Coherent := FALSE;

// Execution projection integrity required.
IF NOT GVL_EXECUTION_PROJECTION_INTEGRITY_FABRIC.Execution_Projection_Integrity_Granted THEN
    L_Integrity_Valid := FALSE;
    L_Error_Code := 52000;
    L_Error_Text := 'Execution projection integrity not granted';
END_IF;

// Governance feedback poisoning detectors.
IF GVL_GOVERNANCE_FEEDBACK_INTEGRITY_FABRIC.Governance_Feedback_Poisoning_Detected THEN
    L_Integrity_Valid := FALSE;
    L_Error_Code := 52001;
    L_Error_Text := 'Governance feedback poisoning detected';
END_IF;

IF GVL_GOVERNANCE_FEEDBACK_INTEGRITY_FABRIC.Execution_Telemetry_Authority_Corruption THEN
    L_Integrity_Valid := FALSE;
    L_Error_Code := 52002;
    L_Error_Text := 'Execution telemetry authority corruption detected';
END_IF;

IF GVL_GOVERNANCE_FEEDBACK_INTEGRITY_FABRIC.CrossEpoch_Feedback_Lineage_Drift THEN
    L_Integrity_Valid := FALSE;
    L_Error_Code := 52003;
    L_Error_Text := 'Cross-epoch feedback lineage drift detected';
END_IF;

IF GVL_GOVERNANCE_FEEDBACK_INTEGRITY_FABRIC.Retroactive_Governance_Mutation_Detected THEN
    L_Integrity_Valid := FALSE;
    L_Error_Code := 52004;
    L_Error_Text := 'Retroactive governance mutation detected';
END_IF;

IF GVL_GOVERNANCE_FEEDBACK_INTEGRITY_FABRIC.Distributed_Feedback_Fork_Detected THEN
    L_Integrity_Valid := FALSE;
    L_Error_Code := 52005;
    L_Error_Text := 'Distributed feedback fork detected';
END_IF;

IF GVL_GOVERNANCE_FEEDBACK_INTEGRITY_FABRIC.Untrusted_Execution_Observation_Injected THEN
    L_Integrity_Valid := FALSE;
    L_Error_Code := 52006;
    L_Error_Text := 'Untrusted execution observation injected';
END_IF;

// Governance feedback validation.
IF L_Integrity_Valid
AND NOT GVL_GOVERNANCE_FEEDBACK_INTEGRITY_FABRIC.Authenticated_Execution_Observation_Valid THEN
    L_Integrity_Valid := FALSE;
    L_Error_Code := 52010;
    L_Error_Text := 'Authenticated execution observation invalid';
END_IF;

IF L_Integrity_Valid
AND NOT GVL_GOVERNANCE_FEEDBACK_INTEGRITY_FABRIC.CrossEpoch_Feedback_Continuity_Stable THEN
    L_Integrity_Valid := FALSE;
    L_Error_Code := 52011;
    L_Error_Text := 'Cross-epoch feedback continuity invalid';
END_IF;

IF L_Integrity_Valid
AND NOT GVL_GOVERNANCE_FEEDBACK_INTEGRITY_FABRIC.Governance_Input_Causality_Grounded THEN
    L_Integrity_Valid := FALSE;
    L_Error_Code := 52012;
    L_Error_Text := 'Governance input causality invalid';
END_IF;

IF L_Integrity_Valid
AND NOT GVL_GOVERNANCE_FEEDBACK_INTEGRITY_FABRIC.Distributed_Feedback_Consensus_Valid THEN
    L_Integrity_Valid := FALSE;
    L_Error_Code := 52013;
    L_Error_Text := 'Distributed feedback consensus invalid';
END_IF;

IF L_Integrity_Valid THEN
    GVL_GOVERNANCE_FEEDBACK_INTEGRITY_FABRIC.Governance_Feedback_Integrity_Valid := TRUE;
    GVL_GOVERNANCE_FEEDBACK_INTEGRITY_FABRIC.Governance_Feedback_Integrity_Granted := TRUE;
    GVL_GOVERNANCE_FEEDBACK_INTEGRITY_FABRIC.Governance_Feedback_Integrity_Quarantine_Active := FALSE;

    GVL_GOVERNANCE_FEEDBACK_INTEGRITY_FABRIC.Execution_Feedback_Causality_Isolated := TRUE;
    GVL_GOVERNANCE_FEEDBACK_INTEGRITY_FABRIC.Governance_Derivation_Inputs_Canonical := TRUE;
    GVL_GOVERNANCE_FEEDBACK_INTEGRITY_FABRIC.Telemetry_To_Authority_Lineage_Valid := TRUE;
    GVL_GOVERNANCE_FEEDBACK_INTEGRITY_FABRIC.Feedback_Epoch_Integrity_Stable := TRUE;
    GVL_GOVERNANCE_FEEDBACK_INTEGRITY_FABRIC.Governance_Feedback_Lineage_Coherent := TRUE;

    GVL_GOVERNANCE_FEEDBACK_INTEGRITY_FABRIC.Governance_Feedback_Integrity_Epoch :=
        GVL_EXECUTION_PROJECTION_INTEGRITY_FABRIC.Execution_Projection_Integrity_Epoch;

    GVL_GOVERNANCE_FEEDBACK_INTEGRITY_FABRIC.Governance_Feedback_Integrity_Epoch_Coherent := TRUE;

    GVL_GOVERNANCE_FEEDBACK_INTEGRITY_FABRIC.Governance_Feedback_Integrity_Last_Update_MS :=
        L_Now_MS;

    GVL_GOVERNANCE_FEEDBACK_INTEGRITY_FABRIC.Governance_Feedback_Integrity_Lease_Expired := FALSE;

    GVL_GOVERNANCE_FEEDBACK_INTEGRITY_FABRIC.Governance_Feedback_Integrity_Last_Error_Code := 0;
    GVL_GOVERNANCE_FEEDBACK_INTEGRITY_FABRIC.Governance_Feedback_Integrity_Last_Error_Text := '';
ELSE
    GVL_GOVERNANCE_FEEDBACK_INTEGRITY_FABRIC.Governance_Feedback_Integrity_Valid := FALSE;
    GVL_GOVERNANCE_FEEDBACK_INTEGRITY_FABRIC.Governance_Feedback_Integrity_Granted := FALSE;
    GVL_GOVERNANCE_FEEDBACK_INTEGRITY_FABRIC.Governance_Feedback_Integrity_Quarantine_Active := TRUE;

    GVL_GOVERNANCE_FEEDBACK_INTEGRITY_FABRIC.Governance_Feedback_Integrity_Lease_Expired := TRUE;

    GVL_GOVERNANCE_FEEDBACK_INTEGRITY_FABRIC.Governance_Feedback_Integrity_Last_Error_Code :=
        L_Error_Code;

    GVL_GOVERNANCE_FEEDBACK_INTEGRITY_FABRIC.Governance_Feedback_Integrity_Last_Error_Text :=
        L_Error_Text;

    GVL_GOVERNANCE_FEEDBACK_INTEGRITY_FABRIC.Governance_Feedback_Integrity_Invalidation_Count :=
        GVL_GOVERNANCE_FEEDBACK_INTEGRITY_FABRIC.Governance_Feedback_Integrity_Invalidation_Count + 1;
END_IF;
          
END_PROGRAM

PROGRAM PRG_Energy_Isolation_Causality_Governor

            IF GVL_AUTHORITY_RESURRECTION_BOUNDARY_FABRIC.Authority_Resurrection_Boundary_Valid
AND NOT GVL_ENERGY_ISOLATION_CAUSALITY_FABRIC.Residual_Energy_Leakage_Detected
AND NOT GVL_ENERGY_ISOLATION_CAUSALITY_FABRIC.CrossDomain_Power_Backfeed_Detected
AND NOT GVL_ENERGY_ISOLATION_CAUSALITY_FABRIC.SplitEnergy_Topology_Detected
AND NOT GVL_ENERGY_ISOLATION_CAUSALITY_FABRIC.Unsafe_Energy_Propagation_Detected THEN

    GVL_ENERGY_ISOLATION_CAUSALITY_FABRIC.Energy_Isolation_Causality_Valid := TRUE;
    GVL_ENERGY_ISOLATION_CAUSALITY_FABRIC.Energy_Isolation_Causality_Granted := TRUE;
    GVL_ENERGY_ISOLATION_CAUSALITY_FABRIC.Physical_Energy_Isolation_Valid := TRUE;
    GVL_ENERGY_ISOLATION_CAUSALITY_FABRIC.Unsafe_Energy_Propagation_Prevented := TRUE;
    GVL_ENERGY_ISOLATION_CAUSALITY_FABRIC.CrossDomain_Power_Segmentation_Canonical := TRUE;
END_IF;
          
END_PROGRAM

PROGRAM PRG_Runtime_Assumption_Integrity_Governor

            // PASSIVE ASSUMPTION OBSERVABILITY ONLY

GVL_RUNTIME_ASSUMPTION_INTEGRITY_FABRIC.Runtime_Assumption_Integrity_Observed :=
    GVL_PROOF_CONTINUITY_AUDIT_FABRIC.Proof_Continuity_Observed;

GVL_RUNTIME_ASSUMPTION_INTEGRITY_FABRIC.Runtime_Assumption_Lineage_Coherent := TRUE;
GVL_RUNTIME_ASSUMPTION_INTEGRITY_FABRIC.Runtime_Assumption_Stability_Observed := TRUE;
          
END_PROGRAM

PROGRAM PRG_Safety_Domain

            // SEMANTIC DOMAIN WRAPPER
// PRESERVES ORIGINAL EXECUTION ORDER
// NO EXECUTION SEMANTICS MUTATION

PRG_Safety();
PRG_Safety_Operator();
PRG_Safety_Shutdown();
PRG_Safety_Recovery();

PRG_Physical_SafeState_Lattice_Governor();
PRG_CrossDomain_FailSafe_Closure_Governor();

PRG_Safety_Observability_Truth_Governor();
PRG_Physical_Safety_Projection_Governor();
          
END_PROGRAM

PROGRAM PRG_Temporal_Stability_Governor
  VAR
    L_Now_MS : UDINT;
    L_Stability_Valid : BOOL := TRUE;
    L_Error_Code : UDINT := 0;
    L_Error_Text : STRING(160) := '';
  END_VAR

            L_Now_MS := GVL_STATUS.G_System_Time_MS;
L_Stability_Valid := TRUE;
L_Error_Code := 0;
L_Error_Text := '';

// Fail-safe defaults.
GVL_TEMPORAL_STABILITY.Temporal_Stability_Valid := FALSE;
GVL_TEMPORAL_STABILITY.Temporal_Stability_Granted := FALSE;
GVL_TEMPORAL_STABILITY.Temporal_Stability_Quarantine_Active := TRUE;

GVL_TEMPORAL_STABILITY.Post_Convergence_Stable := FALSE;
GVL_TEMPORAL_STABILITY.No_Oscillation_Detected := FALSE;
GVL_TEMPORAL_STABILITY.No_Relay_Chatter_Detected := FALSE;
GVL_TEMPORAL_STABILITY.Thermal_Slope_Stable := FALSE;
GVL_TEMPORAL_STABILITY.Pressure_Stable := FALSE;
GVL_TEMPORAL_STABILITY.Flow_Stable := FALSE;

// Temporal stability requires completed physical transaction.
IF NOT GVL_PHYSICAL_TRANSACTION.Physical_Transaction_Granted THEN
    L_Stability_Valid := FALSE;
    L_Error_Code := 28000;
    L_Error_Text := 'Physical transaction not granted';
END_IF;

// Start deterministic observation window.
IF L_Stability_Valid
AND NOT GVL_TEMPORAL_STABILITY.Stability_Observation_Window_Active THEN
    GVL_TEMPORAL_STABILITY.Stability_Observation_Window_Active := TRUE;
    GVL_TEMPORAL_STABILITY.Stability_Window_Start_MS := L_Now_MS;
END_IF;

IF GVL_TEMPORAL_STABILITY.Stability_Observation_Window_Active THEN
    GVL_TEMPORAL_STABILITY.Stability_Window_Elapsed_MS :=
        L_Now_MS - GVL_TEMPORAL_STABILITY.Stability_Window_Start_MS;
END_IF;

// Observation window must fully elapse.
IF L_Stability_Valid
AND (GVL_TEMPORAL_STABILITY.Stability_Window_Elapsed_MS <
     GVL_TEMPORAL_STABILITY.Stability_Window_Target_MS) THEN

    L_Stability_Valid := FALSE;
    L_Error_Code := 28001;
    L_Error_Text := 'Temporal observation window not elapsed';
END_IF;

// Delayed instability detection.
IF GVL_TEMPORAL_STABILITY.Post_Convergence_Oscillation_Detected THEN
    L_Stability_Valid := FALSE;
    L_Error_Code := 28002;
    L_Error_Text := 'Post-convergence oscillation detected';
END_IF;

IF GVL_TEMPORAL_STABILITY.Thermal_Inertia_Rebound_Detected THEN
    L_Stability_Valid := FALSE;
    L_Error_Code := 28003;
    L_Error_Text := 'Thermal inertia rebound detected';
END_IF;

IF GVL_TEMPORAL_STABILITY.Pressure_Rebound_Detected THEN
    L_Stability_Valid := FALSE;
    L_Error_Code := 28004;
    L_Error_Text := 'Pressure rebound detected';
END_IF;

IF GVL_TEMPORAL_STABILITY.Relay_Chatter_Detected THEN
    L_Stability_Valid := FALSE;
    L_Error_Code := 28005;
    L_Error_Text := 'Relay chatter detected';
END_IF;

IF GVL_TEMPORAL_STABILITY.Pump_Cavitation_Recovery_Detected THEN
    L_Stability_Valid := FALSE;
    L_Error_Code := 28006;
    L_Error_Text := 'Pump cavitation recovery detected';
END_IF;

IF GVL_TEMPORAL_STABILITY.Delayed_Actuator_Divergence_Detected THEN
    L_Stability_Valid := FALSE;
    L_Error_Code := 28007;
    L_Error_Text := 'Delayed actuator divergence detected';
END_IF;

// Stable physical conditions required.
IF L_Stability_Valid
AND NOT GVL_TEMPORAL_STABILITY.No_Oscillation_Detected THEN
    L_Stability_Valid := FALSE;
    L_Error_Code := 28010;
    L_Error_Text := 'Oscillation-free state not confirmed';
END_IF;

IF L_Stability_Valid
AND NOT GVL_TEMPORAL_STABILITY.No_Relay_Chatter_Detected THEN
    L_Stability_Valid := FALSE;
    L_Error_Code := 28011;
    L_Error_Text := 'Relay chatter-free state not confirmed';
END_IF;

IF L_Stability_Valid
AND NOT GVL_TEMPORAL_STABILITY.Thermal_Slope_Stable THEN
    L_Stability_Valid := FALSE;
    L_Error_Code := 28012;
    L_Error_Text := 'Thermal slope stability missing';
END_IF;

IF L_Stability_Valid
AND NOT GVL_TEMPORAL_STABILITY.Pressure_Stable THEN
    L_Stability_Valid := FALSE;
    L_Error_Code := 28013;
    L_Error_Text := 'Pressure stability missing';
END_IF;

IF L_Stability_Valid
AND NOT GVL_TEMPORAL_STABILITY.Flow_Stable THEN
    L_Stability_Valid := FALSE;
    L_Error_Code := 28014;
    L_Error_Text := 'Flow stability missing';
END_IF;

IF L_Stability_Valid THEN
    GVL_TEMPORAL_STABILITY.Temporal_Stability_Valid := TRUE;
    GVL_TEMPORAL_STABILITY.Temporal_Stability_Granted := TRUE;
    GVL_TEMPORAL_STABILITY.Temporal_Stability_Quarantine_Active := FALSE;

    GVL_TEMPORAL_STABILITY.Post_Convergence_Stable := TRUE;

    GVL_TEMPORAL_STABILITY.Temporal_Stability_Epoch :=
        GVL_PHYSICAL_TRANSACTION.Physical_Transaction_Epoch;

    GVL_TEMPORAL_STABILITY.Temporal_Stability_Epoch_Coherent := TRUE;

    GVL_TEMPORAL_STABILITY.Temporal_Stability_Last_Update_MS :=
        L_Now_MS;

    GVL_TEMPORAL_STABILITY.Temporal_Stability_Lease_Expired := FALSE;

    GVL_TEMPORAL_STABILITY.Temporal_Stability_Last_Error_Code := 0;
    GVL_TEMPORAL_STABILITY.Temporal_Stability_Last_Error_Text := '';
ELSE
    GVL_TEMPORAL_STABILITY.Temporal_Stability_Valid := FALSE;
    GVL_TEMPORAL_STABILITY.Temporal_Stability_Granted := FALSE;
    GVL_TEMPORAL_STABILITY.Temporal_Stability_Quarantine_Active := TRUE;

    GVL_TEMPORAL_STABILITY.Temporal_Stability_Lease_Expired := TRUE;

    GVL_TEMPORAL_STABILITY.Temporal_Stability_Last_Error_Code :=
        L_Error_Code;

    GVL_TEMPORAL_STABILITY.Temporal_Stability_Last_Error_Text :=
        L_Error_Text;

    GVL_TEMPORAL_STABILITY.Temporal_Stability_Invalidation_Count :=
        GVL_TEMPORAL_STABILITY.Temporal_Stability_Invalidation_Count + 1;
END_IF;
          
END_PROGRAM

PROGRAM PRG_Meta_Governance_Governor
  VAR
    L_Now_MS : UDINT;
    L_Meta_Valid : BOOL := TRUE;
    L_Error_Code : UDINT := 0;
    L_Error_Text : STRING(160) := '';
  END_VAR

            L_Now_MS := GVL_STATUS.G_System_Time_MS;
L_Meta_Valid := TRUE;
L_Error_Code := 0;
L_Error_Text := '';

// Fail-safe defaults.
GVL_META_GOVERNANCE_FABRIC.Meta_Governance_Valid := FALSE;
GVL_META_GOVERNANCE_FABRIC.Meta_Governance_Granted := FALSE;
GVL_META_GOVERNANCE_FABRIC.Meta_Governance_Quarantine_Active := TRUE;

GVL_META_GOVERNANCE_FABRIC.Governance_Graph_Acyclic := FALSE;
GVL_META_GOVERNANCE_FABRIC.Authority_Rooting_Valid := FALSE;
GVL_META_GOVERNANCE_FABRIC.Independent_Validation_Preserved := FALSE;
GVL_META_GOVERNANCE_FABRIC.Meta_Consistency_Coherent := FALSE;
GVL_META_GOVERNANCE_FABRIC.Recursive_Trust_Boundaries_Stable := FALSE;

// Epistemic integrity required.
IF NOT GVL_EPISTEMIC_INTEGRITY_FABRIC.Epistemic_Integrity_Granted THEN
    L_Meta_Valid := FALSE;
    L_Error_Code := 45000;
    L_Error_Text := 'Epistemic integrity authority not granted';
END_IF;

// Meta-governance recursion detectors.
IF GVL_META_GOVERNANCE_FABRIC.Recursive_Authority_Dependency_Detected THEN
    L_Meta_Valid := FALSE;
    L_Error_Code := 45001;
    L_Error_Text := 'Recursive authority dependency detected';
END_IF;

IF GVL_META_GOVERNANCE_FABRIC.Circular_Validation_Chain_Detected THEN
    L_Meta_Valid := FALSE;
    L_Error_Code := 45002;
    L_Error_Text := 'Circular validation chain detected';
END_IF;

IF GVL_META_GOVERNANCE_FABRIC.SelfJustifying_Governance_State_Detected THEN
    L_Meta_Valid := FALSE;
    L_Error_Code := 45003;
    L_Error_Text := 'Self-justifying governance state detected';
END_IF;

IF GVL_META_GOVERNANCE_FABRIC.Epistemic_Recursion_Leakage_Detected THEN
    L_Meta_Valid := FALSE;
    L_Error_Code := 45004;
    L_Error_Text := 'Epistemic recursion leakage detected';
END_IF;

IF GVL_META_GOVERNANCE_FABRIC.Authority_Bootstrap_Paradox_Detected THEN
    L_Meta_Valid := FALSE;
    L_Error_Code := 45005;
    L_Error_Text := 'Authority bootstrap paradox detected';
END_IF;

IF GVL_META_GOVERNANCE_FABRIC.Meta_Consistency_Erosion_Detected THEN
    L_Meta_Valid := FALSE;
    L_Error_Code := 45006;
    L_Error_Text := 'Meta-consistency erosion detected';
END_IF;

// Meta-governance consistency validation.
IF L_Meta_Valid
AND NOT GVL_META_GOVERNANCE_FABRIC.Validator_Independence_Valid THEN
    L_Meta_Valid := FALSE;
    L_Error_Code := 45010;
    L_Error_Text := 'Validator independence invalid';
END_IF;

IF L_Meta_Valid
AND NOT GVL_META_GOVERNANCE_FABRIC.CrossLayer_Causality_Grounded THEN
    L_Meta_Valid := FALSE;
    L_Error_Code := 45011;
    L_Error_Text := 'Cross-layer causality grounding invalid';
END_IF;

IF L_Meta_Valid
AND NOT GVL_META_GOVERNANCE_FABRIC.Bootstrap_Validation_Absent THEN
    L_Meta_Valid := FALSE;
    L_Error_Code := 45012;
    L_Error_Text := 'Bootstrap validation absence invalid';
END_IF;

IF L_Meta_Valid
AND NOT GVL_META_GOVERNANCE_FABRIC.SelfReference_Elimination_Valid THEN
    L_Meta_Valid := FALSE;
    L_Error_Code := 45013;
    L_Error_Text := 'Self-reference elimination invalid';
END_IF;

IF L_Meta_Valid THEN
    GVL_META_GOVERNANCE_FABRIC.Meta_Governance_Valid := TRUE;
    GVL_META_GOVERNANCE_FABRIC.Meta_Governance_Granted := TRUE;
    GVL_META_GOVERNANCE_FABRIC.Meta_Governance_Quarantine_Active := FALSE;

    GVL_META_GOVERNANCE_FABRIC.Governance_Graph_Acyclic := TRUE;
    GVL_META_GOVERNANCE_FABRIC.Authority_Rooting_Valid := TRUE;
    GVL_META_GOVERNANCE_FABRIC.Independent_Validation_Preserved := TRUE;
    GVL_META_GOVERNANCE_FABRIC.Meta_Consistency_Coherent := TRUE;
    GVL_META_GOVERNANCE_FABRIC.Recursive_Trust_Boundaries_Stable := TRUE;

    GVL_META_GOVERNANCE_FABRIC.Meta_Governance_Epoch :=
        GVL_EPISTEMIC_INTEGRITY_FABRIC.Epistemic_Integrity_Epoch;

    GVL_META_GOVERNANCE_FABRIC.Meta_Governance_Epoch_Coherent := TRUE;

    GVL_META_GOVERNANCE_FABRIC.Meta_Governance_Last_Update_MS :=
        L_Now_MS;

    GVL_META_GOVERNANCE_FABRIC.Meta_Governance_Lease_Expired := FALSE;

    GVL_META_GOVERNANCE_FABRIC.Meta_Governance_Last_Error_Code := 0;
    GVL_META_GOVERNANCE_FABRIC.Meta_Governance_Last_Error_Text := '';
ELSE
    GVL_META_GOVERNANCE_FABRIC.Meta_Governance_Valid := FALSE;
    GVL_META_GOVERNANCE_FABRIC.Meta_Governance_Granted := FALSE;
    GVL_META_GOVERNANCE_FABRIC.Meta_Governance_Quarantine_Active := TRUE;

    GVL_META_GOVERNANCE_FABRIC.Meta_Governance_Lease_Expired := TRUE;

    GVL_META_GOVERNANCE_FABRIC.Meta_Governance_Last_Error_Code :=
        L_Error_Code;

    GVL_META_GOVERNANCE_FABRIC.Meta_Governance_Last_Error_Text :=
        L_Error_Text;

    GVL_META_GOVERNANCE_FABRIC.Meta_Governance_Invalidation_Count :=
        GVL_META_GOVERNANCE_FABRIC.Meta_Governance_Invalidation_Count + 1;
END_IF;
          
END_PROGRAM

PROGRAM PRG_Input_Processing
  VAR
    L_i : INT;
    L_HumDelta : REAL;
  END_VAR

            GVL_INPUT.IN_Last_Update_MS := GVL_TIME_SERVICE.G_Now_MS;
GVL_INPUT.IN_Source_Valid := GVL_STATUS.G_Is_Active_PLC;

// RESET FLAGS
GVL_INPUT.IN_Validation_Failed := FALSE;
GVL_INPUT.IN_Anomaly_Detected := FALSE;
GVL_INPUT.IN_Validation_Reason := '';
GVL_INPUT.IN_Anomaly_Reason := '';
GVL_INPUT.IN_Last_Invalid_Zone := 0;
GVL_INPUT.IN_Input_Degraded := FALSE;
GVL_INPUT.IN_Sensor_Fault := FALSE;

GVL_INPUT.IN_Min_Zone_Confidence := REAL#1.0;
GVL_INPUT.IN_Worst_Zone := 0;

// ======================================================
// BASE ENVIRONMENT INPUT AGGREGATION
// ======================================================
GVL_INPUT.IN_Outdoor_Temp := GVL_STATE.G_Outdoor_Temp;
GVL_INPUT.IN_Preheat_Request := GVL_STATE.G_Preheat_Request;
GVL_INPUT.IN_Freeze_Request := GVL_STATE.G_Freeze_Request;

FOR L_i := 1 TO GVL_CONSTANTS.C_MAX_ZONES DO
    GVL_INPUT.IN_Room_Temps[L_i] := GVL_STATE.G_Room_Temps[L_i];
    GVL_INPUT.IN_Room_Hum[L_i] := GVL_STATE.G_Room_Hum[L_i];
    GVL_INPUT.IN_Room_CO2[L_i] := GVL_STATE.G_Room_CO2[L_i];

    // ======================================================
    // RANGE VALIDATION
    // ======================================================
    IF (GVL_INPUT.IN_Room_Temps[L_i] < GVL_INPUT_VALIDATION_CONFIG.G_Room_Temp_Min) OR
       (GVL_INPUT.IN_Room_Temps[L_i] > GVL_INPUT_VALIDATION_CONFIG.G_Room_Temp_Max) THEN
        GVL_INPUT.IN_Validation_Failed := TRUE;
        GVL_INPUT.IN_Input_Degraded := TRUE;
        GVL_INPUT.IN_Sensor_Fault := TRUE;
        GVL_INPUT.IN_Validation_Reason := 'Temp out of range';
        GVL_INPUT.IN_Last_Invalid_Zone := L_i;
    END_IF;

    IF (GVL_INPUT.IN_Room_Hum[L_i] < GVL_INPUT_VALIDATION_CONFIG.G_Room_Hum_Min) OR
       (GVL_INPUT.IN_Room_Hum[L_i] > GVL_INPUT_VALIDATION_CONFIG.G_Room_Hum_Max) THEN
        GVL_INPUT.IN_Validation_Failed := TRUE;
        GVL_INPUT.IN_Input_Degraded := TRUE;
        GVL_INPUT.IN_Sensor_Fault := TRUE;
        GVL_INPUT.IN_Validation_Reason := 'Hum out of range';
        GVL_INPUT.IN_Last_Invalid_Zone := L_i;
    END_IF;

    // ======================================================
    // TEMPERATURE QUALITY SEMANTICS
    // ======================================================
    // Temperature confidence/anomaly publication is now sourced from
    // the passive input quality observer. This replaces the old duplicated
    // local spike calculation while preserving GVL_INPUT as the canonical
    // normalized read-model surface.
    IF GVL_INPUT_QUALITY.G_Room_Temp_Quality[L_i].Quality_Visible THEN
        GVL_INPUT.IN_Room_Temp_Confidence[L_i] :=
            GVL_INPUT_QUALITY.G_Room_Temp_Quality[L_i].Confidence;

        IF GVL_INPUT_QUALITY.G_Room_Temp_Quality[L_i].Value_Degraded THEN
            GVL_INPUT.IN_Input_Degraded := TRUE;
            GVL_INPUT.IN_Anomaly_Detected := TRUE;
            GVL_INPUT.IN_Anomaly_Reason :=
                GVL_INPUT_QUALITY.G_Room_Temp_Quality[L_i].Reason_Text;
            GVL_INPUT.IN_Last_Invalid_Zone := L_i;
        END_IF;

        IF NOT GVL_INPUT_QUALITY.G_Room_Temp_Quality[L_i].Value_Valid THEN
            GVL_INPUT.IN_Validation_Failed := TRUE;
            GVL_INPUT.IN_Sensor_Fault := TRUE;
            GVL_INPUT.IN_Validation_Reason :=
                GVL_INPUT_QUALITY.G_Room_Temp_Quality[L_i].Reason_Text;
            GVL_INPUT.IN_Last_Invalid_Zone := L_i;
        END_IF;
    ELSE
        GVL_INPUT.IN_Room_Temp_Confidence[L_i] :=
            GVL_INPUT_VALIDATION_CONFIG.G_Default_Confidence;
    END_IF;

    // ======================================================
    // HUMIDITY QUALITY SEMANTICS
    // ======================================================
    // Humidity still uses the simplified local path because there is no
    // dedicated humidity input-quality observer yet.
    L_HumDelta := ABS(GVL_INPUT.IN_Room_Hum[L_i] - GVL_INPUT.IN_Room_Hum_Prev[L_i]);

    GVL_INPUT.IN_Room_Hum_Confidence[L_i] :=
        GVL_INPUT_VALIDATION_CONFIG.G_Default_Confidence;

    IF L_HumDelta > GVL_INPUT_VALIDATION_CONFIG.G_Room_Hum_Spike_Threshold THEN
        GVL_INPUT.IN_Room_Hum_Confidence[L_i] :=
            GVL_INPUT_VALIDATION_CONFIG.G_Bad_Spike_Confidence;
        GVL_INPUT.IN_Anomaly_Detected := TRUE;
        GVL_INPUT.IN_Anomaly_Reason := 'Hum spike';
    END_IF;

    // ======================================================
    // REPUTATION
    // ======================================================
    IF GVL_INPUT_VALIDATION_CONFIG.G_Enable_Reputation_Learning THEN
        GVL_INPUT.IN_Room_Temp_Reputation[L_i] :=
            GVL_INPUT.IN_Room_Temp_Reputation[L_i] * (REAL#1.0 - GVL_INPUT_VALIDATION_CONFIG.G_Reputation_Learning_Rate) +
            GVL_INPUT.IN_Room_Temp_Confidence[L_i] * GVL_INPUT_VALIDATION_CONFIG.G_Reputation_Learning_Rate;

        GVL_INPUT.IN_Room_Hum_Reputation[L_i] :=
            GVL_INPUT.IN_Room_Hum_Reputation[L_i] * (REAL#1.0 - GVL_INPUT_VALIDATION_CONFIG.G_Reputation_Learning_Rate) +
            GVL_INPUT.IN_Room_Hum_Confidence[L_i] * GVL_INPUT_VALIDATION_CONFIG.G_Reputation_Learning_Rate;

        GVL_INPUT.IN_Room_Temp_Reputation[L_i] :=
            GVL_INPUT.IN_Room_Temp_Reputation[L_i] +
            (REAL#1.0 - GVL_INPUT.IN_Room_Temp_Reputation[L_i]) * GVL_INPUT_VALIDATION_CONFIG.G_Reputation_Recovery_Decay;

        GVL_INPUT.IN_Room_Hum_Reputation[L_i] :=
            GVL_INPUT.IN_Room_Hum_Reputation[L_i] +
            (REAL#1.0 - GVL_INPUT.IN_Room_Hum_Reputation[L_i]) * GVL_INPUT_VALIDATION_CONFIG.G_Reputation_Recovery_Decay;
    END_IF;

    IF GVL_INPUT.IN_Room_Temp_Reputation[L_i] < GVL_INPUT_VALIDATION_CONFIG.G_Min_Sensor_Confidence THEN
        GVL_INPUT.IN_Room_Temp_Reputation[L_i] :=
            GVL_INPUT_VALIDATION_CONFIG.G_Min_Sensor_Confidence;
    END_IF;

    IF GVL_INPUT.IN_Room_Hum_Reputation[L_i] < GVL_INPUT_VALIDATION_CONFIG.G_Min_Sensor_Confidence THEN
        GVL_INPUT.IN_Room_Hum_Reputation[L_i] :=
            GVL_INPUT_VALIDATION_CONFIG.G_Min_Sensor_Confidence;
    END_IF;

    // ======================================================
    // FINAL ZONE CONFIDENCE
    // ======================================================
    GVL_INPUT.IN_Zone_Confidence[L_i] :=
        (GVL_INPUT.IN_Room_Temp_Confidence[L_i] * GVL_INPUT.IN_Room_Temp_Reputation[L_i] +
         GVL_INPUT.IN_Room_Hum_Confidence[L_i] * GVL_INPUT.IN_Room_Hum_Reputation[L_i]) / REAL#2.0;

    IF GVL_INPUT.IN_Zone_Confidence[L_i] < GVL_INPUT.IN_Min_Zone_Confidence THEN
        GVL_INPUT.IN_Min_Zone_Confidence := GVL_INPUT.IN_Zone_Confidence[L_i];
        GVL_INPUT.IN_Worst_Zone := L_i;
    END_IF;

    GVL_INPUT.IN_Room_Temp_Prev[L_i] := GVL_INPUT.IN_Room_Temps[L_i];
    GVL_INPUT.IN_Room_Hum_Prev[L_i] := GVL_INPUT.IN_Room_Hum[L_i];
END_FOR;

// Floor temperatures are normalized on heating-circuit boundaries,
// not generic zone boundaries.
FOR L_i := 1 TO GVL_CONSTANTS.C_MAX_HEATING_CIRCUITS DO
    GVL_INPUT.IN_Floor_Temps[L_i] := GVL_STATE.G_Floor_Temps[L_i];
END_FOR;

// ======================================================
// SAFETY SENSOR INPUT AGGREGATION
// ======================================================
FOR L_i := 1 TO GVL_CONSTANTS.C_MAX_FLOOD_SENSORS DO
    GVL_INPUT.IN_Water_Sensors[L_i] := GVL_STATE.G_Water_Sensors[L_i];
END_FOR;

FOR L_i := 1 TO GVL_CONSTANTS.C_MAX_SMOKE_SENSORS DO
    GVL_INPUT.IN_Smoke_Sensors[L_i] := GVL_STATE.G_Smoke_Sensors[L_i];
END_FOR;

FOR L_i := 1 TO GVL_CONSTANTS.C_MAX_METHANE_SENSORS DO
    GVL_INPUT.IN_Methane_Sensors[L_i] := GVL_STATE.G_Methane_Sensors[L_i];
END_FOR;

FOR L_i := 1 TO GVL_CONSTANTS.C_MAX_CO_SENSORS DO
    GVL_INPUT.IN_CO_Sensors[L_i] := GVL_STATE.G_CO_Sensors[L_i];
END_FOR;

// >>> BULK_SYNC_ANCHOR: PRG_Input_Processing <<<
          
END_PROGRAM

PROGRAM PRG_Residual_Energy_State_Governor

            IF GVL_ENERGY_ISOLATION_CAUSALITY_FABRIC.Energy_Isolation_Causality_Granted
AND NOT GVL_RESIDUAL_ENERGY_STATE_FABRIC.Latent_Unsafe_Actuation_Detected
AND NOT GVL_RESIDUAL_ENERGY_STATE_FABRIC.Residual_Energy_Persistence_Detected
AND NOT GVL_RESIDUAL_ENERGY_STATE_FABRIC.Unsafe_Thermal_Energy_Retention THEN

    GVL_RESIDUAL_ENERGY_STATE_FABRIC.Residual_Energy_State_Valid := TRUE;
    GVL_RESIDUAL_ENERGY_STATE_FABRIC.Residual_Energy_Bounded := TRUE;
    GVL_RESIDUAL_ENERGY_STATE_FABRIC.Residual_Actuation_Energy_Safe := TRUE;
    GVL_RESIDUAL_ENERGY_STATE_FABRIC.Thermal_Energy_Dissipation_Stable := TRUE;
END_IF;
          
END_PROGRAM

PROGRAM PRG_Distributed_Safety_Reality_Consensus_Governor

            IF GVL_UNSAFE_TRANSITION_FORENSICS_FABRIC.Unsafe_Transition_Forensics_Granted
AND NOT GVL_DISTRIBUTED_SAFETY_REALITY_CONSENSUS_FABRIC.Distributed_Safety_State_Fork
AND NOT GVL_DISTRIBUTED_SAFETY_REALITY_CONSENSUS_FABRIC.Cluster_Safety_Projection_Drift
AND NOT GVL_DISTRIBUTED_SAFETY_REALITY_CONSENSUS_FABRIC.Distributed_Unsafe_State_Hidden THEN

    GVL_DISTRIBUTED_SAFETY_REALITY_CONSENSUS_FABRIC.Distributed_Safety_Reality_Consensus_Valid := TRUE;
    GVL_DISTRIBUTED_SAFETY_REALITY_CONSENSUS_FABRIC.Distributed_Safety_Reality_Consensus_Granted := TRUE;
    GVL_DISTRIBUTED_SAFETY_REALITY_CONSENSUS_FABRIC.Distributed_Safety_Consensus_Valid := TRUE;
    GVL_DISTRIBUTED_SAFETY_REALITY_CONSENSUS_FABRIC.Cluster_Safety_Reality_Stable := TRUE;
    GVL_DISTRIBUTED_SAFETY_REALITY_CONSENSUS_FABRIC.Distributed_Observability_Reality_Equivalence := TRUE;
END_IF;
          
END_PROGRAM

PROGRAM PRG_System_Diagnostics
  VAR
    fbStateTraceLog : FB_State_Trace_Log;
    fbAdapt : FB_Behavior_Adapt;
    fbSystemDiagnosticsPublisher : FB_System_Diagnostics_Publisher;
    L_Pumps_4 : ARRAY[1..4] OF BOOL;
    L_Manifold_Pump_Out_Of_Service : ARRAY[1..GVL_CONSTANTS.C_MAX_MANIFOLDS] OF BOOL;
    L_i : INT;
    L_Last_State_Trace_MS : UDINT;
    L_Hum : REAL;
    L_PrevHum : REAL;
    L_DeltaHum : REAL;
    L_Confidence : REAL;
  END_VAR

            FOR L_i := 1 TO 4 DO
    L_Pumps_4[L_i] := GVL_HEATING_OUTPUT.DO_Manifold_Pumps[L_i];
END_FOR;

FOR L_i := 1 TO GVL_CONSTANTS.C_MAX_MANIFOLDS DO
    L_Manifold_Pump_Out_Of_Service[L_i] := NOT GVL_CONFIG.G_Manifold_Pump_In_Service;
END_FOR;

fbStateTraceLog(
    VI_System_Time := GVL_TIME_SERVICE.G_Now_MS,
    VI_Gas_Alarm := GVL_HEALTH_BRIDGE.G_Gas_Detected OR GVL_HEALTH_BRIDGE.G_CO_Alarm_Level,
    VI_Leak_Alarm := GVL_HEALTH_BRIDGE.G_Leak_Detected,
    VI_Pumps := L_Pumps_4,
    VO_Last_Change_Time => L_Last_State_Trace_MS
);

FOR L_i := 1 TO GVL_CONSTANTS.C_MAX_ZONES DO

    L_Hum := 0.0;

    IF GVL_BEHAVIOR_ADAPT.G_Prev_Valid[L_i] THEN
        L_PrevHum := GVL_BEHAVIOR_ADAPT.G_Prev_Humidity[L_i];
    ELSE
        L_PrevHum := L_Hum;
    END_IF;

    L_DeltaHum := L_PrevHum - L_Hum;

    IF ABS(L_DeltaHum) < 0.5 THEN
        L_Confidence := 0.2;
    ELSE
        L_Confidence := 1.0;
    END_IF;

    IF GVL_INTENT_BEHAVIOR.I_Request_Ventilation_Boost THEN
        fbAdapt(
            iScenario := REASON_SCENARIO_VENT_BOOST,
            iSuccess := (L_DeltaHum > 5.0),
            iMeasuredValue := L_Hum,
            iZone := L_i,
            iConfidence := L_Confidence
        );
    END_IF;

    GVL_BEHAVIOR_ADAPT.G_Prev_Humidity[L_i] := L_Hum;
    GVL_BEHAVIOR_ADAPT.G_Prev_Valid[L_i] := TRUE;

END_FOR;

IF GVL_INTENT_BEHAVIOR.I_Request_Night_Mode THEN
    fbAdapt(
        iScenario := REASON_SCENARIO_NIGHT,
        iSuccess := TRUE,
        iMeasuredValue := 0.0,
        iZone := 0,
        iConfidence := 1.0
    );
END_IF;

fbSystemDiagnosticsPublisher(
    VI_Enable := TRUE,
    VI_System_Time_MS := GVL_TIME_SERVICE.G_Now_MS,
    VI_Backup_Pump_Out_Of_Service := NOT GVL_CONFIG.G_Backup_Circulation_Pump_In_Service,
    VI_Electric_Heater_Out_Of_Service := NOT GVL_CONFIG.G_Electric_Heater_In_Service,
    VI_Manifold_Pump_Out_Of_Service := L_Manifold_Pump_Out_Of_Service,
    VI_DHW_Heating_Pump_Out_Of_Service := NOT GVL_CONFIG.G_DHW_Heating_Pump_In_Service,
    VI_DHW_Circ_Pump_Out_Of_Service := NOT GVL_CONFIG.G_DHW_Circ_Pump_In_Service,
    VI_User_Access_Level := GVL_COMMAND.CMD_User_Access_Level,
    VI_Dangerous_Action_Pending := GVL_COMMAND.CMD_Dangerous_Action_Request,
    VI_Dangerous_Action_Text := 'Dangerous action confirmation requested',
    VI_Sensor_Fault := GVL_STATE.G_Heating_Sensor_Fault OR GVL_STATE.G_DHW_Sensor_Fault,
    VI_IO_Offline := GVL_STATE.G_Heating_IO_Fault OR GVL_STATE.G_DHW_IO_Fault,
    VI_Subsystem_Degraded := GVL_STATE.G_Heating_Subsystem_Degraded OR GVL_STATE.G_DHW_Subsystem_Degraded,
    VI_Manifold_Pressure_Fault := GVL_HEATING_DIAGNOSTICS.G_Manifold_Pressure_Fault,
    VI_Manifold_Current_Fault := GVL_HEATING_DIAGNOSTICS.G_Manifold_Current_Fault,
    VI_Manifold_Return_Temp_Fault := GVL_HEATING_DIAGNOSTICS.G_Manifold_Return_Temp_Fault
);

GVL_System_Diagnostics_Publication.G_System_Diagnostics := fbSystemDiagnosticsPublisher.VO_Diagnostics;
GVL_System_Diagnostics_Publication.G_System_Diagnostics_Publication_Valid := fbSystemDiagnosticsPublisher.VO_Publication_Valid;
GVL_System_Diagnostics_Publication.G_System_Diagnostics_Status_Code := fbSystemDiagnosticsPublisher.VO_Status_Code;
GVL_System_Diagnostics_Publication.G_System_Diagnostics_Status_Text := fbSystemDiagnosticsPublisher.VO_Status_Text;
          
END_PROGRAM

PROGRAM PRG_Trust_Epoch_Monotonicity_Governor
  VAR
    L_Now_MS : UDINT;
    L_Monotonicity_Valid : BOOL := TRUE;
    L_Error_Code : UDINT := 0;
    L_Error_Text : STRING(160) := '';
  END_VAR

            L_Now_MS := GVL_STATUS.G_System_Time_MS;
L_Monotonicity_Valid := TRUE;
L_Error_Code := 0;
L_Error_Text := '';

// Fail-safe defaults.
GVL_TRUST_EPOCH_MONOTONICITY_FABRIC.Trust_Epoch_Monotonicity_Valid := FALSE;
GVL_TRUST_EPOCH_MONOTONICITY_FABRIC.Trust_Epoch_Monotonicity_Granted := FALSE;
GVL_TRUST_EPOCH_MONOTONICITY_FABRIC.Trust_Epoch_Monotonicity_Quarantine_Active := TRUE;

GVL_TRUST_EPOCH_MONOTONICITY_FABRIC.Global_Trust_Epoch_Monotonic := FALSE;
GVL_TRUST_EPOCH_MONOTONICITY_FABRIC.Rollback_Resistant_Authority_Valid := FALSE;
GVL_TRUST_EPOCH_MONOTONICITY_FABRIC.Recovery_Epoch_Strictly_Newer := FALSE;
GVL_TRUST_EPOCH_MONOTONICITY_FABRIC.Distributed_Trust_Vector_Coherent := FALSE;
GVL_TRUST_EPOCH_MONOTONICITY_FABRIC.Irreversible_Trust_Progression_Stable := FALSE;

// Provenance continuity required.
IF NOT GVL_PROVENANCE_CONTINUITY_FABRIC.Provenance_Continuity_Granted THEN
    L_Monotonicity_Valid := FALSE;
    L_Error_Code := 48000;
    L_Error_Text := 'Provenance continuity not granted';
END_IF;

// Temporal trust rollback detectors.
IF GVL_TRUST_EPOCH_MONOTONICITY_FABRIC.Temporal_Trust_Rollback_Detected THEN
    L_Monotonicity_Valid := FALSE;
    L_Error_Code := 48001;
    L_Error_Text := 'Temporal trust rollback detected';
END_IF;

IF GVL_TRUST_EPOCH_MONOTONICITY_FABRIC.Replay_Authority_Epoch_Detected THEN
    L_Monotonicity_Valid := FALSE;
    L_Error_Code := 48002;
    L_Error_Text := 'Replay authority epoch detected';
END_IF;

IF GVL_TRUST_EPOCH_MONOTONICITY_FABRIC.CrossNode_Trust_Vector_Regression THEN
    L_Monotonicity_Valid := FALSE;
    L_Error_Code := 48003;
    L_Error_Text := 'Cross-node trust vector regression detected';
END_IF;

IF GVL_TRUST_EPOCH_MONOTONICITY_FABRIC.Stale_Federation_Epoch_Rejoin THEN
    L_Monotonicity_Valid := FALSE;
    L_Error_Code := 48004;
    L_Error_Text := 'Stale federation epoch rejoin detected';
END_IF;

IF GVL_TRUST_EPOCH_MONOTONICITY_FABRIC.Recovery_Timeline_Fork_Detected THEN
    L_Monotonicity_Valid := FALSE;
    L_Error_Code := 48005;
    L_Error_Text := 'Recovery timeline fork detected';
END_IF;

IF GVL_TRUST_EPOCH_MONOTONICITY_FABRIC.Revoked_Epoch_Resurrection_Detected THEN
    L_Monotonicity_Valid := FALSE;
    L_Error_Code := 48006;
    L_Error_Text := 'Revoked epoch resurrection detected';
END_IF;

// Monotonic trust validation.
IF L_Monotonicity_Valid
AND NOT GVL_TRUST_EPOCH_MONOTONICITY_FABRIC.CrossNode_Trust_Epoch_Aligned THEN
    L_Monotonicity_Valid := FALSE;
    L_Error_Code := 48010;
    L_Error_Text := 'Cross-node trust epoch alignment invalid';
END_IF;

IF L_Monotonicity_Valid
AND NOT GVL_TRUST_EPOCH_MONOTONICITY_FABRIC.Recovery_Timeline_Dominance_Valid THEN
    L_Monotonicity_Valid := FALSE;
    L_Error_Code := 48011;
    L_Error_Text := 'Recovery timeline dominance invalid';
END_IF;

IF L_Monotonicity_Valid
AND NOT GVL_TRUST_EPOCH_MONOTONICITY_FABRIC.Federation_Epoch_Progression_Coherent THEN
    L_Monotonicity_Valid := FALSE;
    L_Error_Code := 48012;
    L_Error_Text := 'Federation epoch progression invalid';
END_IF;

IF L_Monotonicity_Valid
AND NOT GVL_TRUST_EPOCH_MONOTONICITY_FABRIC.Trust_Revocation_History_Monotonic THEN
    L_Monotonicity_Valid := FALSE;
    L_Error_Code := 48013;
    L_Error_Text := 'Trust revocation history monotonicity invalid';
END_IF;

IF L_Monotonicity_Valid THEN
    GVL_TRUST_EPOCH_MONOTONICITY_FABRIC.Trust_Epoch_Monotonicity_Valid := TRUE;
    GVL_TRUST_EPOCH_MONOTONICITY_FABRIC.Trust_Epoch_Monotonicity_Granted := TRUE;
    GVL_TRUST_EPOCH_MONOTONICITY_FABRIC.Trust_Epoch_Monotonicity_Quarantine_Active := FALSE;

    GVL_TRUST_EPOCH_MONOTONICITY_FABRIC.Global_Trust_Epoch_Monotonic := TRUE;
    GVL_TRUST_EPOCH_MONOTONICITY_FABRIC.Rollback_Resistant_Authority_Valid := TRUE;
    GVL_TRUST_EPOCH_MONOTONICITY_FABRIC.Recovery_Epoch_Strictly_Newer := TRUE;
    GVL_TRUST_EPOCH_MONOTONICITY_FABRIC.Distributed_Trust_Vector_Coherent := TRUE;
    GVL_TRUST_EPOCH_MONOTONICITY_FABRIC.Irreversible_Trust_Progression_Stable := TRUE;

    GVL_TRUST_EPOCH_MONOTONICITY_FABRIC.Trust_Epoch_Monotonicity_Epoch :=
        GVL_PROVENANCE_CONTINUITY_FABRIC.Provenance_Continuity_Epoch;

    GVL_TRUST_EPOCH_MONOTONICITY_FABRIC.Trust_Epoch_Monotonicity_Epoch_Coherent := TRUE;

    GVL_TRUST_EPOCH_MONOTONICITY_FABRIC.Trust_Epoch_Monotonicity_Last_Update_MS :=
        L_Now_MS;

    GVL_TRUST_EPOCH_MONOTONICITY_FABRIC.Trust_Epoch_Monotonicity_Lease_Expired := FALSE;

    GVL_TRUST_EPOCH_MONOTONICITY_FABRIC.Trust_Epoch_Monotonicity_Last_Error_Code := 0;
    GVL_TRUST_EPOCH_MONOTONICITY_FABRIC.Trust_Epoch_Monotonicity_Last_Error_Text := '';
ELSE
    GVL_TRUST_EPOCH_MONOTONICITY_FABRIC.Trust_Epoch_Monotonicity_Valid := FALSE;
    GVL_TRUST_EPOCH_MONOTONICITY_FABRIC.Trust_Epoch_Monotonicity_Granted := FALSE;
    GVL_TRUST_EPOCH_MONOTONICITY_FABRIC.Trust_Epoch_Monotonicity_Quarantine_Active := TRUE;

    GVL_TRUST_EPOCH_MONOTONICITY_FABRIC.Trust_Epoch_Monotonicity_Lease_Expired := TRUE;

    GVL_TRUST_EPOCH_MONOTONICITY_FABRIC.Trust_Epoch_Monotonicity_Last_Error_Code :=
        L_Error_Code;

    GVL_TRUST_EPOCH_MONOTONICITY_FABRIC.Trust_Epoch_Monotonicity_Last_Error_Text :=
        L_Error_Text;

    GVL_TRUST_EPOCH_MONOTONICITY_FABRIC.Trust_Epoch_Monotonicity_Invalidation_Count :=
        GVL_TRUST_EPOCH_MONOTONICITY_FABRIC.Trust_Epoch_Monotonicity_Invalidation_Count + 1;
END_IF;
          
END_PROGRAM

PROGRAM PRG_Physical_Safety_Projection_Governor

            IF GVL_SAFETY_OBSERVABILITY_TRUTH_FABRIC.Safety_Observability_Truth_Granted
AND NOT GVL_PHYSICAL_SAFETY_PROJECTION_FABRIC.Physical_Safety_Projection_Drift_Detected
AND NOT GVL_PHYSICAL_SAFETY_PROJECTION_FABRIC.Hidden_Unsafe_Physical_State_Detected
AND NOT GVL_PHYSICAL_SAFETY_PROJECTION_FABRIC.Unsafe_Projection_Backfill_Detected THEN

    GVL_PHYSICAL_SAFETY_PROJECTION_FABRIC.Physical_Safety_Projection_Valid := TRUE;
    GVL_PHYSICAL_SAFETY_PROJECTION_FABRIC.Physical_Safety_Projection_Granted := TRUE;
    GVL_PHYSICAL_SAFETY_PROJECTION_FABRIC.Physical_Plant_Safety_Projection_Stable := TRUE;
    GVL_PHYSICAL_SAFETY_PROJECTION_FABRIC.Energy_State_Safety_Projection_Valid := TRUE;
    GVL_PHYSICAL_SAFETY_PROJECTION_FABRIC.Recovery_State_Safety_Projection_Valid := TRUE;
END_IF;
          
END_PROGRAM

PROGRAM PRG_OpenTherm_Transport
  VAR
    L_i : INT;
    L_Status_Word : WORD;
    L_Heartbeat : UDINT;
    L_Ack_Seq : UDINT;
  END_VAR

            // ======================================================
// REAL TRANSPORT LAYER CONTRACT
// ======================================================
// This layer converts high-level command/status structures
// into transport-safe wire images.
//
// Real Modbus RTU/TCP or serial IO code must:
//   1. Write G_Wire_Image command fields to adapter registers.
//   2. Read adapter status registers into G_Wire_Image status fields.
//
// This program keeps protocol encoding/decoding centralized.
// It does not claim transport online unless OpenTherm is enabled.
// ======================================================

IF NOT GVL_CONFIG.G_OpenTherm_Enabled THEN
    GVL_OPENTHERM_ADAPTER.G_Transport_Online := FALSE;
    GVL_OPENTHERM_ADAPTER.G_Transport_Error := FALSE;

    FOR L_i := 1 TO GVL_CONSTANTS.C_MAX_BOILERS DO
        GVL_OPENTHERM_ADAPTER.G_Wire_Image[L_i].Cmd_Enable := 0;
        GVL_OPENTHERM_ADAPTER.G_Wire_Image[L_i].Cmd_Setpoint_x10 := 0;
        GVL_OPENTHERM_ADAPTER.G_Wire_Image[L_i].Cmd_Seq_Lo := 0;
        GVL_OPENTHERM_ADAPTER.G_Wire_Image[L_i].Cmd_Seq_Hi := 0;

        GVL_OPENTHERM_ADAPTER.G_Status[L_i].Raw_Online := FALSE;
        GVL_OPENTHERM_ADAPTER.G_Status[L_i].Raw_Error := FALSE;
        GVL_OPENTHERM_ADAPTER.G_Status[L_i].Raw_Flame := FALSE;
        GVL_OPENTHERM_ADAPTER.G_Status[L_i].Raw_Status_Word := 0;
    END_FOR;

    RETURN;
END_IF;

GVL_OPENTHERM_ADAPTER.G_Transport_Online := TRUE;
GVL_OPENTHERM_ADAPTER.G_Transport_Error := FALSE;
GVL_OPENTHERM_ADAPTER.G_Last_Transport_Update_MS := GVL_STATUS.G_System_Time_MS;

FOR L_i := 1 TO GVL_CONSTANTS.C_MAX_BOILERS DO

    // ======================================================
    // COMMAND → WIRE IMAGE
    // ======================================================
    IF GVL_OPENTHERM_ADAPTER.G_Command[L_i].Enable THEN
        GVL_OPENTHERM_ADAPTER.G_Wire_Image[L_i].Cmd_Enable := 1;
    ELSE
        GVL_OPENTHERM_ADAPTER.G_Wire_Image[L_i].Cmd_Enable := 0;
    END_IF;

    GVL_OPENTHERM_ADAPTER.G_Wire_Image[L_i].Cmd_Setpoint_x10 :=
        GVL_OPENTHERM_ADAPTER.G_Command[L_i].Setpoint_x10;

    GVL_OPENTHERM_ADAPTER.G_Wire_Image[L_i].Cmd_Seq_Lo :=
        UDINT_TO_WORD(GVL_OPENTHERM_ADAPTER.G_Command[L_i].Sequence AND 16#FFFF);

    GVL_OPENTHERM_ADAPTER.G_Wire_Image[L_i].Cmd_Seq_Hi :=
        UDINT_TO_WORD(SHR(GVL_OPENTHERM_ADAPTER.G_Command[L_i].Sequence, 16));

    // ======================================================
    // WIRE IMAGE → STATUS
    // ======================================================
    L_Heartbeat :=
        WORD_TO_UDINT(GVL_OPENTHERM_ADAPTER.G_Wire_Image[L_i].Status_Heartbeat_Lo)
        OR SHL(
            WORD_TO_UDINT(GVL_OPENTHERM_ADAPTER.G_Wire_Image[L_i].Status_Heartbeat_Hi),
            16
        );

    L_Ack_Seq :=
        WORD_TO_UDINT(GVL_OPENTHERM_ADAPTER.G_Wire_Image[L_i].Status_Ack_Seq_Lo)
        OR SHL(
            WORD_TO_UDINT(GVL_OPENTHERM_ADAPTER.G_Wire_Image[L_i].Status_Ack_Seq_Hi),
            16
        );

    GVL_OPENTHERM_ADAPTER.G_Status[L_i].Raw_Heartbeat := L_Heartbeat;
    GVL_OPENTHERM_ADAPTER.G_Status[L_i].Raw_Ack_Seq := L_Ack_Seq;

    L_Status_Word :=
        GVL_OPENTHERM_ADAPTER.G_Wire_Image[L_i].Status_Word;

    GVL_OPENTHERM_ADAPTER.G_Status[L_i].Raw_Online :=
        (L_Status_Word AND 16#0001) <> 0;

    GVL_OPENTHERM_ADAPTER.G_Status[L_i].Raw_Error :=
        (L_Status_Word AND 16#0002) <> 0;

    GVL_OPENTHERM_ADAPTER.G_Status[L_i].Raw_Flame :=
        (L_Status_Word AND 16#0004) <> 0;

    GVL_OPENTHERM_ADAPTER.G_Status[L_i].Raw_Status_Word :=
        L_Status_Word;

    GVL_OPENTHERM_ADAPTER.G_Status[L_i].Raw_Error_Code :=
        GVL_OPENTHERM_ADAPTER.G_Wire_Image[L_i].Error_Code;

    GVL_OPENTHERM_ADAPTER.G_Status[L_i].Raw_Modulation_x10 :=
        GVL_OPENTHERM_ADAPTER.G_Wire_Image[L_i].Modulation_x10;

    GVL_OPENTHERM_ADAPTER.G_Status[L_i].Raw_Boiler_Temp_x10 :=
        WORD_TO_INT(GVL_OPENTHERM_ADAPTER.G_Wire_Image[L_i].Boiler_Temp_x10);

END_FOR;
          
END_PROGRAM

PROGRAM PRG_Provenance_Continuity_Governor
  VAR
    L_Now_MS : UDINT;
    L_Continuity_Valid : BOOL := TRUE;
    L_Error_Code : UDINT := 0;
    L_Error_Text : STRING(160) := '';
  END_VAR

            L_Now_MS := GVL_STATUS.G_System_Time_MS;
L_Continuity_Valid := TRUE;
L_Error_Code := 0;
L_Error_Text := '';

// Fail-safe defaults.
GVL_PROVENANCE_CONTINUITY_FABRIC.Provenance_Continuity_Valid := FALSE;
GVL_PROVENANCE_CONTINUITY_FABRIC.Provenance_Continuity_Granted := FALSE;
GVL_PROVENANCE_CONTINUITY_FABRIC.Provenance_Continuity_Quarantine_Active := TRUE;

GVL_PROVENANCE_CONTINUITY_FABRIC.Recovery_Provenance_Reattested := FALSE;
GVL_PROVENANCE_CONTINUITY_FABRIC.Authority_Resurrection_Authentic := FALSE;
GVL_PROVENANCE_CONTINUITY_FABRIC.Federation_Rejoin_Provenance_Valid := FALSE;
GVL_PROVENANCE_CONTINUITY_FABRIC.PostRecovery_TrustSeed_Coherent := FALSE;
GVL_PROVENANCE_CONTINUITY_FABRIC.CrossEpoch_Provenance_Continuity_Stable := FALSE;

// Authority provenance required.
IF NOT GVL_AUTHORITY_PROVENANCE_FABRIC.Authority_Provenance_Granted THEN
    L_Continuity_Valid := FALSE;
    L_Error_Code := 47000;
    L_Error_Text := 'Authority provenance not granted';
END_IF;

// Post-recovery provenance bypass detectors.
IF GVL_PROVENANCE_CONTINUITY_FABRIC.Stale_Provenance_Resurrection_Detected THEN
    L_Continuity_Valid := FALSE;
    L_Error_Code := 47001;
    L_Error_Text := 'Stale provenance resurrection detected';
END_IF;

IF GVL_PROVENANCE_CONTINUITY_FABRIC.Recovered_Authority_Without_Reattestation_Detected THEN
    L_Continuity_Valid := FALSE;
    L_Error_Code := 47002;
    L_Error_Text := 'Recovered authority without re-attestation detected';
END_IF;

IF GVL_PROVENANCE_CONTINUITY_FABRIC.Federation_Rejoin_Without_Provenance_Detected THEN
    L_Continuity_Valid := FALSE;
    L_Error_Code := 47003;
    L_Error_Text := 'Federation rejoin without provenance detected';
END_IF;

IF GVL_PROVENANCE_CONTINUITY_FABRIC.CrossEpoch_Trust_Continuity_Broken THEN
    L_Continuity_Valid := FALSE;
    L_Error_Code := 47004;
    L_Error_Text := 'Cross-epoch trust continuity broken';
END_IF;

IF GVL_PROVENANCE_CONTINUITY_FABRIC.Recovery_Trust_Seed_Drift_Detected THEN
    L_Continuity_Valid := FALSE;
    L_Error_Code := 47005;
    L_Error_Text := 'Recovery trust-seed drift detected';
END_IF;

IF GVL_PROVENANCE_CONTINUITY_FABRIC.Provenance_Resurrection_Bypass_Detected THEN
    L_Continuity_Valid := FALSE;
    L_Error_Code := 47006;
    L_Error_Text := 'Provenance resurrection bypass detected';
END_IF;

// Provenance continuity validation.
IF L_Continuity_Valid
AND NOT GVL_PROVENANCE_CONTINUITY_FABRIC.Recovery_Epoch_Authenticity_Valid THEN
    L_Continuity_Valid := FALSE;
    L_Error_Code := 47010;
    L_Error_Text := 'Recovery epoch authenticity invalid';
END_IF;

IF L_Continuity_Valid
AND NOT GVL_PROVENANCE_CONTINUITY_FABRIC.Distributed_Rejoin_Attestation_Coherent THEN
    L_Continuity_Valid := FALSE;
    L_Error_Code := 47011;
    L_Error_Text := 'Distributed rejoin attestation invalid';
END_IF;

IF L_Continuity_Valid
AND NOT GVL_PROVENANCE_CONTINUITY_FABRIC.Authority_Restoration_Provenance_Grounded THEN
    L_Continuity_Valid := FALSE;
    L_Error_Code := 47012;
    L_Error_Text := 'Authority restoration provenance invalid';
END_IF;

IF L_Continuity_Valid
AND NOT GVL_PROVENANCE_CONTINUITY_FABRIC.Provenance_Lease_Continuity_Valid THEN
    L_Continuity_Valid := FALSE;
    L_Error_Code := 47013;
    L_Error_Text := 'Provenance lease continuity invalid';
END_IF;

IF L_Continuity_Valid THEN
    GVL_PROVENANCE_CONTINUITY_FABRIC.Provenance_Continuity_Valid := TRUE;
    GVL_PROVENANCE_CONTINUITY_FABRIC.Provenance_Continuity_Granted := TRUE;
    GVL_PROVENANCE_CONTINUITY_FABRIC.Provenance_Continuity_Quarantine_Active := FALSE;

    GVL_PROVENANCE_CONTINUITY_FABRIC.Recovery_Provenance_Reattested := TRUE;
    GVL_PROVENANCE_CONTINUITY_FABRIC.Authority_Resurrection_Authentic := TRUE;
    GVL_PROVENANCE_CONTINUITY_FABRIC.Federation_Rejoin_Provenance_Valid := TRUE;
    GVL_PROVENANCE_CONTINUITY_FABRIC.PostRecovery_TrustSeed_Coherent := TRUE;
    GVL_PROVENANCE_CONTINUITY_FABRIC.CrossEpoch_Provenance_Continuity_Stable := TRUE;

    GVL_PROVENANCE_CONTINUITY_FABRIC.Provenance_Continuity_Epoch :=
        GVL_AUTHORITY_PROVENANCE_FABRIC.Authority_Provenance_Epoch;

    GVL_PROVENANCE_CONTINUITY_FABRIC.Provenance_Continuity_Epoch_Coherent := TRUE;

    GVL_PROVENANCE_CONTINUITY_FABRIC.Provenance_Continuity_Last_Update_MS :=
        L_Now_MS;

    GVL_PROVENANCE_CONTINUITY_FABRIC.Provenance_Continuity_Lease_Expired := FALSE;

    GVL_PROVENANCE_CONTINUITY_FABRIC.Provenance_Continuity_Last_Error_Code := 0;
    GVL_PROVENANCE_CONTINUITY_FABRIC.Provenance_Continuity_Last_Error_Text := '';
ELSE
    GVL_PROVENANCE_CONTINUITY_FABRIC.Provenance_Continuity_Valid := FALSE;
    GVL_PROVENANCE_CONTINUITY_FABRIC.Provenance_Continuity_Granted := FALSE;
    GVL_PROVENANCE_CONTINUITY_FABRIC.Provenance_Continuity_Quarantine_Active := TRUE;

    GVL_PROVENANCE_CONTINUITY_FABRIC.Provenance_Continuity_Lease_Expired := TRUE;

    GVL_PROVENANCE_CONTINUITY_FABRIC.Provenance_Continuity_Last_Error_Code :=
        L_Error_Code;

    GVL_PROVENANCE_CONTINUITY_FABRIC.Provenance_Continuity_Last_Error_Text :=
        L_Error_Text;

    GVL_PROVENANCE_CONTINUITY_FABRIC.Provenance_Continuity_Invalidation_Count :=
        GVL_PROVENANCE_CONTINUITY_FABRIC.Provenance_Continuity_Invalidation_Count + 1;
END_IF;
          
END_PROGRAM

PROGRAM PRG_CrossDomain_FailSafe_Closure_Governor
  VAR
    L_Now_MS : UDINT;
    L_Valid : BOOL := TRUE;
  END_VAR

            L_Now_MS := GVL_STATUS.G_System_Time_MS;

GVL_CROSSDOMAIN_FAILSAFE_CLOSURE_FABRIC.CrossDomain_FailSafe_Closure_Valid := FALSE;
GVL_CROSSDOMAIN_FAILSAFE_CLOSURE_FABRIC.CrossDomain_FailSafe_Closure_Granted := FALSE;
GVL_CROSSDOMAIN_FAILSAFE_CLOSURE_FABRIC.CrossDomain_FailSafe_Closure_Quarantine_Active := TRUE;

IF NOT GVL_PHYSICAL_SAFESTATE_LATTICE_FABRIC.Physical_SafeState_Lattice_Granted THEN
    L_Valid := FALSE;
END_IF;

IF GVL_CROSSDOMAIN_FAILSAFE_CLOSURE_FABRIC.CrossDomain_FailSafe_Conflict_Detected
OR GVL_CROSSDOMAIN_FAILSAFE_CLOSURE_FABRIC.Unsafe_Recovery_Topology_Detected
OR GVL_CROSSDOMAIN_FAILSAFE_CLOSURE_FABRIC.CrossDomain_Recovery_Race_Detected
OR GVL_CROSSDOMAIN_FAILSAFE_CLOSURE_FABRIC.Distributed_SafeState_Fork_Detected
OR GVL_CROSSDOMAIN_FAILSAFE_CLOSURE_FABRIC.PowerDomain_Unsafe_Reactivation_Detected
OR GVL_CROSSDOMAIN_FAILSAFE_CLOSURE_FABRIC.MultiDomain_Recovery_Deadlock_Detected THEN
    L_Valid := FALSE;
END_IF;

IF L_Valid THEN
    GVL_CROSSDOMAIN_FAILSAFE_CLOSURE_FABRIC.CrossDomain_FailSafe_Closure_Valid := TRUE;
    GVL_CROSSDOMAIN_FAILSAFE_CLOSURE_FABRIC.CrossDomain_FailSafe_Closure_Granted := TRUE;
    GVL_CROSSDOMAIN_FAILSAFE_CLOSURE_FABRIC.CrossDomain_FailSafe_Closure_Quarantine_Active := FALSE;

    GVL_CROSSDOMAIN_FAILSAFE_CLOSURE_FABRIC.CrossDomain_SafeState_Compatibility_Valid := TRUE;
    GVL_CROSSDOMAIN_FAILSAFE_CLOSURE_FABRIC.FailSafe_Topology_Closure_Canonical := TRUE;
    GVL_CROSSDOMAIN_FAILSAFE_CLOSURE_FABRIC.MultiDomain_SafeTransition_Stable := TRUE;
    GVL_CROSSDOMAIN_FAILSAFE_CLOSURE_FABRIC.SafeState_Recovery_Ordering_Bounded := TRUE;
    GVL_CROSSDOMAIN_FAILSAFE_CLOSURE_FABRIC.Physical_Domain_Isolation_Coherent := TRUE;

    GVL_CROSSDOMAIN_FAILSAFE_CLOSURE_FABRIC.CrossDomain_FailSafe_Closure_Epoch :=
        GVL_PHYSICAL_SAFESTATE_LATTICE_FABRIC.Physical_SafeState_Lattice_Epoch;

    GVL_CROSSDOMAIN_FAILSAFE_CLOSURE_FABRIC.CrossDomain_FailSafe_Closure_Epoch_Coherent := TRUE;
    GVL_CROSSDOMAIN_FAILSAFE_CLOSURE_FABRIC.CrossDomain_FailSafe_Closure_Last_Update_MS := L_Now_MS;
    GVL_CROSSDOMAIN_FAILSAFE_CLOSURE_FABRIC.CrossDomain_FailSafe_Closure_Lease_Expired := FALSE;
END_IF;
          
END_PROGRAM

PROGRAM PRG_Runtime_Sustainability_Governor
  VAR
    L_Now_MS : UDINT;
    L_Runtime_Valid : BOOL := TRUE;
    L_Error_Code : UDINT := 0;
    L_Error_Text : STRING(160) := '';
  END_VAR

            L_Now_MS := GVL_STATUS.G_System_Time_MS;
L_Runtime_Valid := TRUE;
L_Error_Code := 0;
L_Error_Text := '';

// Fail-safe defaults.
GVL_RUNTIME_SUSTAINABILITY_FABRIC.Runtime_Sustainability_Valid := FALSE;
GVL_RUNTIME_SUSTAINABILITY_FABRIC.Runtime_Sustainability_Granted := FALSE;
GVL_RUNTIME_SUSTAINABILITY_FABRIC.Runtime_Sustainability_Quarantine_Active := TRUE;

GVL_RUNTIME_SUSTAINABILITY_FABRIC.Deterministic_Cycle_Budget_Stable := FALSE;
GVL_RUNTIME_SUSTAINABILITY_FABRIC.Runtime_Queue_Load_Stable := FALSE;
GVL_RUNTIME_SUSTAINABILITY_FABRIC.Memory_Fragmentation_Stable := FALSE;
GVL_RUNTIME_SUSTAINABILITY_FABRIC.Watchdog_Jitter_Stable := FALSE;
GVL_RUNTIME_SUSTAINABILITY_FABRIC.HA_Synchronization_Load_Stable := FALSE;

// Energy causality authority required.
IF NOT GVL_ENERGY_CAUSALITY_FABRIC.Energy_Causality_Granted THEN
    L_Runtime_Valid := FALSE;
    L_Error_Code := 38000;
    L_Error_Text := 'Energy causality authority not granted';
END_IF;

// Resource-collapse detectors.
IF GVL_RUNTIME_SUSTAINABILITY_FABRIC.Memory_Fragmentation_Drift_Detected THEN
    L_Runtime_Valid := FALSE;
    L_Error_Code := 38001;
    L_Error_Text := 'Memory fragmentation drift detected';
END_IF;

IF GVL_RUNTIME_SUSTAINABILITY_FABRIC.Queue_Saturation_Detected THEN
    L_Runtime_Valid := FALSE;
    L_Error_Code := 38002;
    L_Error_Text := 'Runtime queue saturation detected';
END_IF;

IF GVL_RUNTIME_SUSTAINABILITY_FABRIC.Historical_Persistence_Amplification_Detected THEN
    L_Runtime_Valid := FALSE;
    L_Error_Code := 38003;
    L_Error_Text := 'Historical persistence amplification detected';
END_IF;

IF GVL_RUNTIME_SUSTAINABILITY_FABRIC.Watchdog_Jitter_Escalation_Detected THEN
    L_Runtime_Valid := FALSE;
    L_Error_Code := 38004;
    L_Error_Text := 'Watchdog jitter escalation detected';
END_IF;

IF GVL_RUNTIME_SUSTAINABILITY_FABRIC.HASynchronization_Overload_Detected THEN
    L_Runtime_Valid := FALSE;
    L_Error_Code := 38005;
    L_Error_Text := 'HA synchronization overload detected';
END_IF;

IF GVL_RUNTIME_SUSTAINABILITY_FABRIC.Deterministic_Cycle_Erosion_Detected THEN
    L_Runtime_Valid := FALSE;
    L_Error_Code := 38006;
    L_Error_Text := 'Deterministic cycle erosion detected';
END_IF;

// Long-term runtime sustainability validation.
IF L_Runtime_Valid
AND NOT GVL_RUNTIME_SUSTAINABILITY_FABRIC.Historical_Persistence_Load_Stable THEN
    L_Runtime_Valid := FALSE;
    L_Error_Code := 38010;
    L_Error_Text := 'Historical persistence load unstable';
END_IF;

IF L_Runtime_Valid
AND NOT GVL_RUNTIME_SUSTAINABILITY_FABRIC.Snapshot_Publication_Stable THEN
    L_Runtime_Valid := FALSE;
    L_Error_Code := 38011;
    L_Error_Text := 'Snapshot publication unstable';
END_IF;

IF L_Runtime_Valid
AND NOT GVL_RUNTIME_SUSTAINABILITY_FABRIC.Distributed_Runtime_Load_Coherent THEN
    L_Runtime_Valid := FALSE;
    L_Error_Code := 38012;
    L_Error_Text := 'Distributed runtime load coherence invalid';
END_IF;

IF L_Runtime_Valid
AND NOT GVL_RUNTIME_SUSTAINABILITY_FABRIC.Runtime_Evolution_Sustainable THEN
    L_Runtime_Valid := FALSE;
    L_Error_Code := 38013;
    L_Error_Text := 'Runtime evolution sustainability invalid';
END_IF;

IF L_Runtime_Valid THEN
    GVL_RUNTIME_SUSTAINABILITY_FABRIC.Runtime_Sustainability_Valid := TRUE;
    GVL_RUNTIME_SUSTAINABILITY_FABRIC.Runtime_Sustainability_Granted := TRUE;
    GVL_RUNTIME_SUSTAINABILITY_FABRIC.Runtime_Sustainability_Quarantine_Active := FALSE;

    GVL_RUNTIME_SUSTAINABILITY_FABRIC.Deterministic_Cycle_Budget_Stable := TRUE;
    GVL_RUNTIME_SUSTAINABILITY_FABRIC.Runtime_Queue_Load_Stable := TRUE;
    GVL_RUNTIME_SUSTAINABILITY_FABRIC.Memory_Fragmentation_Stable := TRUE;
    GVL_RUNTIME_SUSTAINABILITY_FABRIC.Watchdog_Jitter_Stable := TRUE;
    GVL_RUNTIME_SUSTAINABILITY_FABRIC.HA_Synchronization_Load_Stable := TRUE;

    GVL_RUNTIME_SUSTAINABILITY_FABRIC.Runtime_Sustainability_Epoch :=
        GVL_ENERGY_CAUSALITY_FABRIC.Energy_Causality_Epoch;

    GVL_RUNTIME_SUSTAINABILITY_FABRIC.Runtime_Sustainability_Epoch_Coherent := TRUE;

    GVL_RUNTIME_SUSTAINABILITY_FABRIC.Runtime_Sustainability_Last_Update_MS :=
        L_Now_MS;

    GVL_RUNTIME_SUSTAINABILITY_FABRIC.Runtime_Sustainability_Lease_Expired := FALSE;

    GVL_RUNTIME_SUSTAINABILITY_FABRIC.Runtime_Sustainability_Last_Error_Code := 0;
    GVL_RUNTIME_SUSTAINABILITY_FABRIC.Runtime_Sustainability_Last_Error_Text := '';
ELSE
    GVL_RUNTIME_SUSTAINABILITY_FABRIC.Runtime_Sustainability_Valid := FALSE;
    GVL_RUNTIME_SUSTAINABILITY_FABRIC.Runtime_Sustainability_Granted := FALSE;
    GVL_RUNTIME_SUSTAINABILITY_FABRIC.Runtime_Sustainability_Quarantine_Active := TRUE;

    GVL_RUNTIME_SUSTAINABILITY_FABRIC.Runtime_Sustainability_Lease_Expired := TRUE;

    GVL_RUNTIME_SUSTAINABILITY_FABRIC.Runtime_Sustainability_Last_Error_Code :=
        L_Error_Code;

    GVL_RUNTIME_SUSTAINABILITY_FABRIC.Runtime_Sustainability_Last_Error_Text :=
        L_Error_Text;

    GVL_RUNTIME_SUSTAINABILITY_FABRIC.Runtime_Sustainability_Invalidation_Count :=
        GVL_RUNTIME_SUSTAINABILITY_FABRIC.Runtime_Sustainability_Invalidation_Count + 1;
END_IF;
          
END_PROGRAM

PROGRAM PRG_Distributed_Commit_Ingestion

            // ======================================================
// DISTRIBUTED COMMIT INGESTION
// ======================================================
// Explicit peer distributed commit ingestion layer.
//
// Purpose:
// normalize replicated peer commit-handshake state into
// distributed commit peer-input fields.
//
// This layer does NOT:
// - perform commit reconciliation
// - validate replay continuity
// - validate peer acknowledgements
// ======================================================

IF GVL_HA_SESSION_REPLICATION.HA_Remote_Session_Valid THEN
    GVL_DISTRIBUTED_COMMIT.Peer_Publication_Commit_Epoch :=
        GVL_HA_SESSION_REPLICATION.HA_Remote_Publication_Commit_Epoch;

    GVL_DISTRIBUTED_COMMIT.Peer_Prepare_Epoch :=
        GVL_HA_SESSION_REPLICATION.HA_Remote_Prepare_Epoch;

    GVL_DISTRIBUTED_COMMIT.Peer_Commit_Ack_Valid :=
        GVL_HA_SESSION_REPLICATION.HA_Remote_Commit_Ack_Valid;

    GVL_DISTRIBUTED_COMMIT.Peer_Commit_Last_Refresh_MS :=
        GVL_HA_SESSION_REPLICATION.HA_Remote_Commit_Last_Refresh_MS;
ELSE
    GVL_DISTRIBUTED_COMMIT.Peer_Publication_Commit_Epoch := 0;
    GVL_DISTRIBUTED_COMMIT.Peer_Prepare_Epoch := 0;
    GVL_DISTRIBUTED_COMMIT.Peer_Commit_Ack_Valid := FALSE;
    GVL_DISTRIBUTED_COMMIT.Peer_Commit_Last_Refresh_MS := 0;
END_IF;

// >>> BULK_SYNC_ANCHOR: PRG_Distributed_Commit_Ingestion <<<
          
END_PROGRAM

PROGRAM PRG_Execution_Projection_Integrity_Governor
  VAR
    L_Now_MS : UDINT;
    L_Integrity_Valid : BOOL := TRUE;
    L_Error_Code : UDINT := 0;
    L_Error_Text : STRING(160) := '';
  END_VAR

            L_Now_MS := GVL_STATUS.G_System_Time_MS;
L_Integrity_Valid := TRUE;
L_Error_Code := 0;
L_Error_Text := '';

// Fail-safe defaults.
GVL_EXECUTION_PROJECTION_INTEGRITY_FABRIC.Execution_Projection_Integrity_Valid := FALSE;
GVL_EXECUTION_PROJECTION_INTEGRITY_FABRIC.Execution_Projection_Integrity_Granted := FALSE;
GVL_EXECUTION_PROJECTION_INTEGRITY_FABRIC.Execution_Projection_Integrity_Quarantine_Active := TRUE;

GVL_EXECUTION_PROJECTION_INTEGRITY_FABRIC.Execution_Authority_Projection_Consistent := FALSE;
GVL_EXECUTION_PROJECTION_INTEGRITY_FABRIC.CrossDomain_Actuation_Enforcement_Aligned := FALSE;
GVL_EXECUTION_PROJECTION_INTEGRITY_FABRIC.Physical_Execution_Governance_Canonical := FALSE;
GVL_EXECUTION_PROJECTION_INTEGRITY_FABRIC.Actuation_Surface_Consensus_Valid := FALSE;
GVL_EXECUTION_PROJECTION_INTEGRITY_FABRIC.Execution_Projection_Lineage_Coherent := FALSE;

// Governance observer consensus required.
IF NOT GVL_GOVERNANCE_OBSERVER_CONSENSUS_FABRIC.Governance_Observer_Consensus_Granted THEN
    L_Integrity_Valid := FALSE;
    L_Error_Code := 51000;
    L_Error_Text := 'Governance observer consensus not granted';
END_IF;

// Execution projection split-brain detectors.
IF GVL_EXECUTION_PROJECTION_INTEGRITY_FABRIC.Execution_Projection_Divergence_Detected THEN
    L_Integrity_Valid := FALSE;
    L_Error_Code := 51001;
    L_Error_Text := 'Execution projection divergence detected';
END_IF;

IF GVL_EXECUTION_PROJECTION_INTEGRITY_FABRIC.Actuation_Path_Authority_Bypass_Detected THEN
    L_Integrity_Valid := FALSE;
    L_Error_Code := 51002;
    L_Error_Text := 'Actuation path authority bypass detected';
END_IF;

IF GVL_EXECUTION_PROJECTION_INTEGRITY_FABRIC.CrossDomain_Enforcement_Fork_Detected THEN
    L_Integrity_Valid := FALSE;
    L_Error_Code := 51003;
    L_Error_Text := 'Cross-domain enforcement fork detected';
END_IF;

IF GVL_EXECUTION_PROJECTION_INTEGRITY_FABRIC.Canonical_Governance_Execution_Lost THEN
    L_Integrity_Valid := FALSE;
    L_Error_Code := 51004;
    L_Error_Text := 'Canonical governance execution lost';
END_IF;

IF GVL_EXECUTION_PROJECTION_INTEGRITY_FABRIC.Runtime_Execution_Lineage_Drift_Detected THEN
    L_Integrity_Valid := FALSE;
    L_Error_Code := 51005;
    L_Error_Text := 'Runtime execution lineage drift detected';
END_IF;

IF GVL_EXECUTION_PROJECTION_INTEGRITY_FABRIC.Distributed_Actuation_Reality_Fork_Detected THEN
    L_Integrity_Valid := FALSE;
    L_Error_Code := 51006;
    L_Error_Text := 'Distributed actuation reality fork detected';
END_IF;

// Execution enforcement validation.
IF L_Integrity_Valid
AND NOT GVL_EXECUTION_PROJECTION_INTEGRITY_FABRIC.Runtime_Actuation_Projection_Stable THEN
    L_Integrity_Valid := FALSE;
    L_Error_Code := 51010;
    L_Error_Text := 'Runtime actuation projection invalid';
END_IF;

IF L_Integrity_Valid
AND NOT GVL_EXECUTION_PROJECTION_INTEGRITY_FABRIC.Distributed_Execution_Equivalence_Valid THEN
    L_Integrity_Valid := FALSE;
    L_Error_Code := 51011;
    L_Error_Text := 'Distributed execution equivalence invalid';
END_IF;

IF L_Integrity_Valid
AND NOT GVL_EXECUTION_PROJECTION_INTEGRITY_FABRIC.Execution_Governance_Causality_Grounded THEN
    L_Integrity_Valid := FALSE;
    L_Error_Code := 51012;
    L_Error_Text := 'Execution governance causality invalid';
END_IF;

IF L_Integrity_Valid
AND NOT GVL_EXECUTION_PROJECTION_INTEGRITY_FABRIC.Physical_Enforcement_Timeline_Monotonic THEN
    L_Integrity_Valid := FALSE;
    L_Error_Code := 51013;
    L_Error_Text := 'Physical enforcement timeline monotonicity invalid';
END_IF;

IF L_Integrity_Valid THEN
    GVL_EXECUTION_PROJECTION_INTEGRITY_FABRIC.Execution_Projection_Integrity_Valid := TRUE;
    GVL_EXECUTION_PROJECTION_INTEGRITY_FABRIC.Execution_Projection_Integrity_Granted := TRUE;
    GVL_EXECUTION_PROJECTION_INTEGRITY_FABRIC.Execution_Projection_Integrity_Quarantine_Active := FALSE;

    GVL_EXECUTION_PROJECTION_INTEGRITY_FABRIC.Execution_Authority_Projection_Consistent := TRUE;
    GVL_EXECUTION_PROJECTION_INTEGRITY_FABRIC.CrossDomain_Actuation_Enforcement_Aligned := TRUE;
    GVL_EXECUTION_PROJECTION_INTEGRITY_FABRIC.Physical_Execution_Governance_Canonical := TRUE;
    GVL_EXECUTION_PROJECTION_INTEGRITY_FABRIC.Actuation_Surface_Consensus_Valid := TRUE;
    GVL_EXECUTION_PROJECTION_INTEGRITY_FABRIC.Execution_Projection_Lineage_Coherent := TRUE;

    GVL_EXECUTION_PROJECTION_INTEGRITY_FABRIC.Execution_Projection_Integrity_Epoch :=
        GVL_GOVERNANCE_OBSERVER_CONSENSUS_FABRIC.Governance_Observer_Consensus_Epoch;

    GVL_EXECUTION_PROJECTION_INTEGRITY_FABRIC.Execution_Projection_Integrity_Epoch_Coherent := TRUE;

    GVL_EXECUTION_PROJECTION_INTEGRITY_FABRIC.Execution_Projection_Integrity_Last_Update_MS :=
        L_Now_MS;

    GVL_EXECUTION_PROJECTION_INTEGRITY_FABRIC.Execution_Projection_Integrity_Lease_Expired := FALSE;

    GVL_EXECUTION_PROJECTION_INTEGRITY_FABRIC.Execution_Projection_Integrity_Last_Error_Code := 0;
    GVL_EXECUTION_PROJECTION_INTEGRITY_FABRIC.Execution_Projection_Integrity_Last_Error_Text := '';
ELSE
    GVL_EXECUTION_PROJECTION_INTEGRITY_FABRIC.Execution_Projection_Integrity_Valid := FALSE;
    GVL_EXECUTION_PROJECTION_INTEGRITY_FABRIC.Execution_Projection_Integrity_Granted := FALSE;
    GVL_EXECUTION_PROJECTION_INTEGRITY_FABRIC.Execution_Projection_Integrity_Quarantine_Active := TRUE;

    GVL_EXECUTION_PROJECTION_INTEGRITY_FABRIC.Execution_Projection_Integrity_Lease_Expired := TRUE;

    GVL_EXECUTION_PROJECTION_INTEGRITY_FABRIC.Execution_Projection_Integrity_Last_Error_Code :=
        L_Error_Code;

    GVL_EXECUTION_PROJECTION_INTEGRITY_FABRIC.Execution_Projection_Integrity_Last_Error_Text :=
        L_Error_Text;

    GVL_EXECUTION_PROJECTION_INTEGRITY_FABRIC.Execution_Projection_Integrity_Invalidation_Count :=
        GVL_EXECUTION_PROJECTION_INTEGRITY_FABRIC.Execution_Projection_Integrity_Invalidation_Count + 1;
END_IF;
          
END_PROGRAM

PROGRAM PRG_Config_Versioning
  VAR
    L_i : INT;
    L_Config_Error : BOOL;
  END_VAR

            // Detect config error from validation layer
L_Config_Error := GVL_STATUS.G_Diagnostics.Sensor_Fault OR GVL_STATUS.G_Diagnostics.Subsystem_Degraded;

// --- Save snapshot when system is healthy ---
IF NOT L_Config_Error THEN
    FOR L_i := 1 TO GVL_CONSTANTS.C_MAX_HEATING_CIRCUITS DO
        GVL_CONFIG_BACKUP.G_Backup_FloorHeating_Configs[L_i] := GVL_CONFIG.G_HMI_FloorHeating_Configs[L_i];
    END_FOR;

    GVL_CONFIG_BACKUP.G_Backup_Max_Active_Manifolds := GVL_CONFIG.G_Max_Active_Manifolds;
    GVL_CONFIG_BACKUP.G_Backup_Max_Thermal_Budget := GVL_CONFIG.G_Max_Thermal_Budget;

    GVL_CONFIG_BACKUP.G_Backup_Valid := TRUE;
END_IF;

// --- Rollback if config invalid ---
IF L_Config_Error THEN

    // Freeze system via command layer
    GVL_COMMAND_SHADOW.G_Heating_Block := TRUE;
    GVL_COMMAND_SHADOW.G_Boiler_Stop := TRUE;

    // Restore snapshot only if valid
    IF GVL_CONFIG_BACKUP.G_Backup_Valid THEN
        FOR L_i := 1 TO GVL_CONSTANTS.C_MAX_HEATING_CIRCUITS DO
            GVL_CONFIG.G_HMI_FloorHeating_Configs[L_i] := GVL_CONFIG_BACKUP.G_Backup_FloorHeating_Configs[L_i];
        END_FOR;

        GVL_CONFIG.G_Max_Active_Manifolds := GVL_CONFIG_BACKUP.G_Backup_Max_Active_Manifolds;
        GVL_CONFIG.G_Max_Thermal_Budget := GVL_CONFIG_BACKUP.G_Backup_Max_Thermal_Budget;

        GVL_STATUS.G_System_Mode_Text := 'CONFIG ROLLBACK';
    ELSE
        GVL_STATUS.G_System_Mode_Text := 'CONFIG INVALID - NO BACKUP';
    END_IF;
END_IF;

// >>> BULK_SYNC_ANCHOR: PRG_Config_Versioning <<<
          
END_PROGRAM

PROGRAM PRG_Governance_Publication_Binding_Governor
  VAR
    L_Now_MS : UDINT;
    L_Valid : BOOL := TRUE;
    L_Error_Code : UDINT := 0;
    L_Error_Text : STRING(160) := '';
  END_VAR

            L_Now_MS := GVL_STATUS.G_System_Time_MS;
L_Valid := TRUE;
L_Error_Code := 0;
L_Error_Text := '';

// Fail-safe defaults.
GVL_GOVERNANCE_PUBLICATION_BINDING_FABRIC.Governance_Publication_Binding_Valid := FALSE;
GVL_GOVERNANCE_PUBLICATION_BINDING_FABRIC.Governance_Publication_Binding_Granted := FALSE;
GVL_GOVERNANCE_PUBLICATION_BINDING_FABRIC.Governance_Publication_Binding_Quarantine_Active := TRUE;

GVL_GOVERNANCE_PUBLICATION_BINDING_FABRIC.Observability_Publication_Causality_Valid := FALSE;
GVL_GOVERNANCE_PUBLICATION_BINDING_FABRIC.Upstream_Governance_Lease_Fresh := FALSE;
GVL_GOVERNANCE_PUBLICATION_BINDING_FABRIC.Governance_Publication_Epoch_Coherent := FALSE;
GVL_GOVERNANCE_PUBLICATION_BINDING_FABRIC.Publication_Quarantine_Propagation_Valid := FALSE;
GVL_GOVERNANCE_PUBLICATION_BINDING_FABRIC.Canonical_Observability_Reality_Consistent := FALSE;

// Governance liveness integrity required.
IF NOT GVL_GOVERNANCE_LIVENESS_INTEGRITY_FABRIC.Governance_Liveness_Integrity_Granted THEN
    L_Valid := FALSE;
    L_Error_Code := 55000;
    L_Error_Text := 'Governance liveness integrity not granted';
END_IF;

// Publication binding detectors.
IF GVL_GOVERNANCE_PUBLICATION_BINDING_FABRIC.Stale_Valid_Publication_Detected THEN
    L_Valid := FALSE;
    L_Error_Code := 55001;
    L_Error_Text := 'Stale valid publication detected';
END_IF;

IF GVL_GOVERNANCE_PUBLICATION_BINDING_FABRIC.LeaseExpired_Governance_Published_As_Healthy THEN
    L_Valid := FALSE;
    L_Error_Code := 55002;
    L_Error_Text := 'Lease-expired governance published as healthy';
END_IF;

IF GVL_GOVERNANCE_PUBLICATION_BINDING_FABRIC.Quarantine_State_Publication_Bypass THEN
    L_Valid := FALSE;
    L_Error_Code := 55003;
    L_Error_Text := 'Quarantine state publication bypass';
END_IF;

IF GVL_GOVERNANCE_PUBLICATION_BINDING_FABRIC.Governance_Invalidation_Hidden_From_Observability THEN
    L_Valid := FALSE;
    L_Error_Code := 55004;
    L_Error_Text := 'Governance invalidation hidden from observability';
END_IF;

IF GVL_GOVERNANCE_PUBLICATION_BINDING_FABRIC.Distributed_Publication_State_Fork_Detected THEN
    L_Valid := FALSE;
    L_Error_Code := 55005;
    L_Error_Text := 'Distributed publication state fork detected';
END_IF;

IF GVL_GOVERNANCE_PUBLICATION_BINDING_FABRIC.Historical_Invalidation_Causality_Lost THEN
    L_Valid := FALSE;
    L_Error_Code := 55006;
    L_Error_Text := 'Historical invalidation causality lost';
END_IF;

// Publication validation.
IF L_Valid
AND NOT GVL_GOVERNANCE_PUBLICATION_BINDING_FABRIC.Diagnostics_Publication_Consistency_Valid THEN
    L_Valid := FALSE;
    L_Error_Code := 55010;
    L_Error_Text := 'Diagnostics publication consistency invalid';
END_IF;

IF L_Valid
AND NOT GVL_GOVERNANCE_PUBLICATION_BINDING_FABRIC.HMI_Publication_State_Aligned THEN
    L_Valid := FALSE;
    L_Error_Code := 55011;
    L_Error_Text := 'HMI publication state alignment invalid';
END_IF;

IF L_Valid
AND NOT GVL_GOVERNANCE_PUBLICATION_BINDING_FABRIC.Blackbox_Invalidation_Lineage_Valid THEN
    L_Valid := FALSE;
    L_Error_Code := 55012;
    L_Error_Text := 'Blackbox invalidation lineage invalid';
END_IF;

IF L_Valid
AND NOT GVL_GOVERNANCE_PUBLICATION_BINDING_FABRIC.Distributed_Publication_Consensus_Valid THEN
    L_Valid := FALSE;
    L_Error_Code := 55013;
    L_Error_Text := 'Distributed publication consensus invalid';
END_IF;

IF L_Valid THEN
    GVL_GOVERNANCE_PUBLICATION_BINDING_FABRIC.Governance_Publication_Binding_Valid := TRUE;
    GVL_GOVERNANCE_PUBLICATION_BINDING_FABRIC.Governance_Publication_Binding_Granted := TRUE;
    GVL_GOVERNANCE_PUBLICATION_BINDING_FABRIC.Governance_Publication_Binding_Quarantine_Active := FALSE;

    GVL_GOVERNANCE_PUBLICATION_BINDING_FABRIC.Observability_Publication_Causality_Valid := TRUE;
    GVL_GOVERNANCE_PUBLICATION_BINDING_FABRIC.Upstream_Governance_Lease_Fresh := TRUE;
    GVL_GOVERNANCE_PUBLICATION_BINDING_FABRIC.Governance_Publication_Epoch_Coherent := TRUE;
    GVL_GOVERNANCE_PUBLICATION_BINDING_FABRIC.Publication_Quarantine_Propagation_Valid := TRUE;
    GVL_GOVERNANCE_PUBLICATION_BINDING_FABRIC.Canonical_Observability_Reality_Consistent := TRUE;

    GVL_GOVERNANCE_PUBLICATION_BINDING_FABRIC.Governance_Publication_Binding_Epoch :=
        GVL_GOVERNANCE_LIVENESS_INTEGRITY_FABRIC.Governance_Liveness_Integrity_Epoch;

    GVL_GOVERNANCE_PUBLICATION_BINDING_FABRIC.Governance_Publication_Binding_Epoch_Coherent_Runtime := TRUE;

    GVL_GOVERNANCE_PUBLICATION_BINDING_FABRIC.Governance_Publication_Binding_Last_Update_MS :=
        L_Now_MS;

    GVL_GOVERNANCE_PUBLICATION_BINDING_FABRIC.Governance_Publication_Binding_Lease_Expired := FALSE;

    GVL_GOVERNANCE_PUBLICATION_BINDING_FABRIC.Governance_Publication_Binding_Last_Error_Code := 0;
    GVL_GOVERNANCE_PUBLICATION_BINDING_FABRIC.Governance_Publication_Binding_Last_Error_Text := '';
ELSE
    GVL_GOVERNANCE_PUBLICATION_BINDING_FABRIC.Governance_Publication_Binding_Valid := FALSE;
    GVL_GOVERNANCE_PUBLICATION_BINDING_FABRIC.Governance_Publication_Binding_Granted := FALSE;
    GVL_GOVERNANCE_PUBLICATION_BINDING_FABRIC.Governance_Publication_Binding_Quarantine_Active := TRUE;

    GVL_GOVERNANCE_PUBLICATION_BINDING_FABRIC.Governance_Publication_Binding_Lease_Expired := TRUE;

    GVL_GOVERNANCE_PUBLICATION_BINDING_FABRIC.Governance_Publication_Binding_Last_Error_Code :=
        L_Error_Code;

    GVL_GOVERNANCE_PUBLICATION_BINDING_FABRIC.Governance_Publication_Binding_Last_Error_Text :=
        L_Error_Text;

    GVL_GOVERNANCE_PUBLICATION_BINDING_FABRIC.Governance_Publication_Binding_Invalidation_Count :=
        GVL_GOVERNANCE_PUBLICATION_BINDING_FABRIC.Governance_Publication_Binding_Invalidation_Count + 1;
END_IF;
          
END_PROGRAM

PROGRAM PRG_Security
  VAR
    L_i : INT;
    L_Motion_Sensors_16 : ARRAY[1..16] OF BOOL;
    fbSecurityManager : FB_Security_System_Manager;
    fbAccessControl : FB_Access_Control;
  END_VAR

            FOR L_i := 1 TO 16 DO
    L_Motion_Sensors_16[L_i] := GVL_STATE.G_Motion_Sensors[L_i];
END_FOR;
// 7. Система безопасности (Охранная сигнализация)
fbSecurityManager(
    VI_System_Time_MS := GVL_STATUS.G_System_Time_MS,
    VI_IsActivePLC := GVL_STATUS.G_Is_Active_PLC,
    VI_Motion_Sensors := L_Motion_Sensors_16,
    VI_Door_Sensors := GVL_STATE.G_Door_Sensors,
    VI_Window_Sensors := GVL_STATE.G_Window_Sensors,
    VI_Arm_Request := GVL_INTENT_USER.I_Arm_Request,
    VI_Disarm_Request := GVL_INTENT_USER.I_Disarm_Request,
    VI_PIN_Code := GVL_INTENT_USER.I_PIN_Code,
    VI_RFID_Tag := GVL_INTENT_USER.I_RFID_Tag,
    VI_2FA_Code := GVL_INTENT_USER.I_2FA_Code_In,
    VI_Config := GVL_CONFIG.G_Security_Config,
    VI_Bypass_Motion := GVL_CONFIG.G_Security_Config.bypass_motion,
    VI_Bypass_Doors := GVL_CONFIG.G_Security_Config.bypass_doors,
    VI_Bypass_Windows := GVL_CONFIG.G_Security_Config.bypass_windows,
    VI_Current_TOD := GVL_STATUS.G_Current_TOD,
    VO_Armed => GVL_ALARM.G_Security_Armed,
    VO_Alarm_Active => GVL_ALARM.G_Security_Alarm,
    VO_Siren_Active => GVL_ALARM.G_Security_Siren,
    VO_Status_Msg => GVL_STATUS.G_Security_Status_Msg,
    VO_Send_Code_Req => GVL_COMMAND.G_Send_2FA_Req,
    VO_Code_To_Send => GVL_COMMAND.G_2FA_Code_Out
);

